LIN {X 0,Y 331.929,Z 1000.191,A -85,B 0,C 180,E1 23009.158,E2 23009.158} C_VEL
LIN {X 0,Y 336.667,Z 1013.449,A -85,B 0,C 180,E1 23012.773,E2 23012.773} C_VEL
LIN {X 0,Y 338.095,Z 1019.979,A -85,B 0,C 180,E1 23013.863,E2 23013.863} C_VEL
LIN {X 0,Y 332.466,Z 1050.059,A -85,B 0,C 180,E1 23015.679,E2 23015.679} C_VEL
LIN {X 0,Y 325.019,Z 1075.85,A -85,B 0,C 180,E1 23018.168,E2 23018.168} C_VEL
LIN {X 0,Y 315.792,Z 1098.668,A -85,B 0,C 180,E1 23021.521,E2 23021.521} C_VEL
LIN {X 0,Y 310.988,Z 1108.297,A -85,B 0,C 180,E1 23023.502,E2 23023.502} C_VEL
LIN {X 0,Y 302.321,Z 1118.917,A -85,B 0,C 180,E1 23025.58,E2 23025.58} C_VEL
LIN {X 0,Y 294.454,Z 1126.629,A -85,B 0,C 180,E1 23027.603,E2 23027.603} C_VEL
LIN {X 0,Y 293.706,Z 1127.508,A -85,B 0,C 180,E1 23027.959,E2 23027.959} C_VEL
LIN {X 0,Y 286.319,Z 1135.333,A -85,B 0,C 180,E1 23032.421,E2 23032.421} C_VEL
LIN {X 0,Y 280.665,Z 1138.98,A -85,B 0,C 180,E1 23036.917,E2 23036.917} C_VEL
LIN {X 0,Y 277.782,Z 1139.343,A -85,B 0,C 180,E1 23040.003,E2 23040.003} C_VEL
LIN {X 0,Y 274.693,Z 1136.847,A -85,B 0,C 180,E1 23044.737,E2 23044.737} C_VEL
LIN {X 0,Y 272.966,Z 1127.598,A -85,B 0,C 180,E1 23051.175,E2 23051.175} C_VEL
LIN {X 0,Y 273.213,Z 1112.925,A -85,B 0,C 180,E1 23056.884,E2 23056.884} C_VEL
LIN {X 0,Y 274.614,Z 1092.685,A -85,B 0,C 180,E1 23061.997,E2 23061.997} C_VEL
LIN {X 0,Y 276.602,Z 1068.704,A -85,B 0,C 180,E1 23066.137,E2 23066.137} C_VEL
LIN {X 0,Y 278.792,Z 1039.52,A -85,B 0,C 180,E1 23069.486,E2 23069.486} C_VEL
LIN {X 0,Y 280.451,Z 1007.858,A -85,B 0,C 180,E1 23071.663,E2 23071.663} C_VEL
LIN {X 0,Y 280.123,Z 983.5,A -85,B 0,C 180,E1 23072.673,E2 23072.673} C_VEL
LIN {X 0,Y 267.448,Z 923.03,A -85,B 0,C 180,E1 23075.683,E2 23075.683} C_VEL
LIN {X 0,Y 266.889,Z 923.03,A -85,B 0,C 180,E1 23082.804,E2 23082.804} C_VEL
LIN {X 0,Y 266.968,Z 923.03,A -85,B 0,C 180,E1 23091.46,E2 23091.46} C_VEL
LIN {X 0,Y 267.275,Z 923.03,A -85,B 0,C 180,E1 23099.384,E2 23099.384} C_VEL
LIN {X 0,Y 267.761,Z 923.03,A -85,B 0,C 180,E1 23106.703,E2 23106.703} C_VEL
LIN {X 0,Y 268.363,Z 923.03,A -85,B 0,C 180,E1 23113.62,E2 23113.62} C_VEL
LIN {X 0,Y 269.003,Z 923.03,A -85,B 0,C 180,E1 23120.27,E2 23120.27} C_VEL
LIN {X 0,Y 269.819,Z 923.03,A -85,B 0,C 180,E1 23126.762,E2 23126.762} C_VEL
LIN {X 0,Y 269.811,Z 923.03,A -85,B 0,C 180,E1 23133.182,E2 23133.182} C_VEL
LIN {X 0,Y 269.095,Z 923.03,A -85,B 0,C 180,E1 23139.669,E2 23139.669} C_VEL
LIN {X 0,Y 268.337,Z 923.03,A -85,B 0,C 180,E1 23146.786,E2 23146.786} C_VEL
LIN {X 0,Y 267.656,Z 923.03,A -85,B 0,C 180,E1 23155.396,E2 23155.396} C_VEL
LIN {X 0,Y 267.187,Z 923.03,A -85,B 0,C 180,E1 23164.403,E2 23164.403} C_VEL
LIN {X 0,Y 267.237,Z 923.488,A -85,B 0,C 180,E1 23165.586,E2 23165.586} C_VEL
LIN {X 0,Y 284.856,Z 968.437,A -85,B 0,C 180,E1 23170.572,E2 23170.572} C_VEL
LIN {X 0,Y 296.502,Z 1005.612,A -85,B 0,C 180,E1 23174.909,E2 23174.909} C_VEL
LIN {X 0,Y 304.304,Z 1038.041,A -85,B 0,C 180,E1 23179.036,E2 23179.036} C_VEL
LIN {X 0,Y 295.095,Z 1075.692,A -85,B 0,C 180,E1 23183.463,E2 23183.463} C_VEL
LIN {X 0,Y 286.275,Z 1109.373,A -85,B 0,C 180,E1 23189.022,E2 23189.022} C_VEL
LIN {X 0,Y 279.131,Z 1136.473,A -85,B 0,C 180,E1 23195.19,E2 23195.19} C_VEL
LIN {X 0,Y 274.28,Z 1158.137,A -85,B 0,C 180,E1 23201.943,E2 23201.943} C_VEL
LIN {X 0,Y 271.653,Z 1173.928,A -85,B 0,C 180,E1 23208.77,E2 23208.77} C_VEL
LIN {X 0,Y 270.65,Z 1184.291,A -85,B 0,C 180,E1 23215.193,E2 23215.193} C_VEL
LIN {X 0,Y 270.557,Z 1190.919,A -85,B 0,C 180,E1 23221.597,E2 23221.597} C_VEL
LIN {X 0,Y 272.362,Z 1194.634,A -85,B 0,C 180,E1 23229.578,E2 23229.578} C_VEL
LIN {X 0,Y 278.537,Z 1193.012,A -85,B 0,C 180,E1 23238.993,E2 23238.993} C_VEL
LIN {X 0,Y 290.948,Z 1185.504,A -85,B 0,C 180,E1 23247.864,E2 23247.864} C_VEL
LIN {X 0,Y 311.71,Z 1171.475,A -85,B 0,C 180,E1 23256.283,E2 23256.283} C_VEL
LIN {X 0,Y 339.898,Z 1151.742,A -85,B 0,C 180,E1 23263.248,E2 23263.248} C_VEL
LIN {X 0,Y 340.347,Z 1151.495,A -85,B 0,C 180,E1 23263.626,E2 23263.626} C_VEL
LIN {X 0,Y 309.964,Z 1177.069,A -85,B 0,C 180,E1 23270.708,E2 23270.708} C_VEL
LIN {X 0,Y 288.327,Z 1196.897,A -85,B 0,C 180,E1 23279.408,E2 23279.408} C_VEL
LIN {X 0,Y 276.425,Z 1209.235,A -85,B 0,C 180,E1 23288.32,E2 23288.32} C_VEL
LIN {X 0,Y 271.361,Z 1215.518,A -85,B 0,C 180,E1 23297.16,E2 23297.16} C_VEL
LIN {X 0,Y 270.484,Z 1216.446,A -85,B 0,C 180,E1 23303.614,E2 23303.614} C_VEL
LIN {X 0,Y 271.033,Z 1214.048,A -85,B 0,C 180,E1 23310.028,E2 23310.028} C_VEL
LIN {X 0,Y 271.147,Z 1206.707,A -85,B 0,C 180,E1 23317.231,E2 23317.231} C_VEL
LIN {X 0,Y 272.139,Z 1193.796,A -85,B 0,C 180,E1 23324.501,E2 23324.501} C_VEL
LIN {X 0,Y 275.469,Z 1175.838,A -85,B 0,C 180,E1 23332.023,E2 23332.023} C_VEL
LIN {X 0,Y 281.759,Z 1158.597,A -85,B 0,C 180,E1 23338.405,E2 23338.405} C_VEL
LIN {X 0,Y 290.902,Z 1135.195,A -85,B 0,C 180,E1 23344.184,E2 23344.184} C_VEL
LIN {X 0,Y 301.149,Z 1107.507,A -85,B 0,C 180,E1 23348.871,E2 23348.871} C_VEL
LIN {X 0,Y 310.736,Z 1076.284,A -85,B 0,C 180,E1 23352.52,E2 23352.52} C_VEL
LIN {X 0,Y 318.06,Z 1045.689,A -85,B 0,C 180,E1 23354.842,E2 23354.842} C_VEL
LIN {X 0,Y 321.177,Z 1017.496,A -85,B 0,C 180,E1 23359.484,E2 23359.484} C_VEL
LIN {X 0,Y 325.671,Z 998.479,A -85,B 0,C 180,E1 23362.748,E2 23362.748} C_VEL
LIN {X 0,Y 326.577,Z 1000.295,A -85,B 0,C 180,E1 23364.99,E2 23364.99} C_VEL
LIN {X 0,Y 329.513,Z 1007.381,A -85,B 0,C 180,E1 23368.754,E2 23368.754} C_VEL
LIN {X 0,Y 333.618,Z 1020.084,A -85,B 0,C 180,E1 23372.232,E2 23372.232} C_VEL
LIN {X 0,Y 334.133,Z 1023.713,A -85,B 0,C 180,E1 23372.802,E2 23372.802} C_VEL
LIN {X 0,Y 327.641,Z 1054.65,A -85,B 0,C 180,E1 23374.772,E2 23374.772} C_VEL
LIN {X 0,Y 319.445,Z 1080.19,A -85,B 0,C 180,E1 23377.386,E2 23377.386} C_VEL
LIN {X 0,Y 309.736,Z 1101.939,A -85,B 0,C 180,E1 23380.776,E2 23380.776} C_VEL
LIN {X 0,Y 299.636,Z 1119.417,A -85,B 0,C 180,E1 23385.025,E2 23385.025} C_VEL
LIN {X 0,Y 293.706,Z 1127.508,A -85,B 0,C 180,E1 23387.959,E2 23387.959} C_VEL
LIN {X 0,Y 285,Z 1134.232,A -85,B 0,C 180,E1 23390.669,E2 23390.669} C_VEL
LIN {X 0,Y 276.923,Z 1138.639,A -85,B 0,C 180,E1 23393.437,E2 23393.437} C_VEL
LIN {X 0,Y 276.615,Z 1138.783,A -85,B 0,C 180,E1 23393.649,E2 23393.649} C_VEL
LIN {X 0,Y 272.435,Z 1140.471,A -85,B 0,C 180,E1 23397.182,E2 23397.182} C_VEL
LIN {X 0,Y 267.601,Z 1138.671,A -85,B 0,C 180,E1 23403.241,E2 23403.241} C_VEL
LIN {X 0,Y 265.203,Z 1130.248,A -85,B 0,C 180,E1 23409.846,E2 23409.846} C_VEL
LIN {X 0,Y 265.193,Z 1116.066,A -85,B 0,C 180,E1 23415.884,E2 23415.884} C_VEL
LIN {X 0,Y 266.366,Z 1096.688,A -85,B 0,C 180,E1 23421.21,E2 23421.21} C_VEL
LIN {X 0,Y 268.449,Z 1072.024,A -85,B 0,C 180,E1 23425.77,E2 23425.77} C_VEL
LIN {X 0,Y 270.68,Z 1043.898,A -85,B 0,C 180,E1 23429.244,E2 23429.244} C_VEL
LIN {X 0,Y 272.452,Z 1012.551,A -85,B 0,C 180,E1 23431.636,E2 23431.636} C_VEL
LIN {X 0,Y 272.442,Z 985.065,A -85,B 0,C 180,E1 23432.86,E2 23432.86} C_VEL
LIN {X 0,Y 259.474,Z 923.03,A -85,B 0,C 180,E1 23436.06,E2 23436.06} C_VEL
LIN {X 0,Y 258.804,Z 923.03,A -85,B 0,C 180,E1 23445.485,E2 23445.485} C_VEL
LIN {X 0,Y 259.146,Z 923.03,A -85,B 0,C 180,E1 23454.727,E2 23454.727} C_VEL
LIN {X 0,Y 259.491,Z 923.03,A -85,B 0,C 180,E1 23462.203,E2 23462.203} C_VEL
LIN {X 0,Y 260.037,Z 923.03,A -85,B 0,C 180,E1 23469.565,E2 23469.565} C_VEL
LIN {X 0,Y 260.736,Z 923.03,A -85,B 0,C 180,E1 23476.567,E2 23476.567} C_VEL
LIN {X 0,Y 261.406,Z 923.03,A -85,B 0,C 180,E1 23483.332,E2 23483.332} C_VEL
LIN {X 0,Y 262.275,Z 923.03,A -85,B 0,C 180,E1 23489.971,E2 23489.971} C_VEL
LIN {X 0,Y 261.431,Z 923.03,A -85,B 0,C 180,E1 23496.608,E2 23496.608} C_VEL
LIN {X 0,Y 260.78,Z 923.03,A -85,B 0,C 180,E1 23503.371,E2 23503.371} C_VEL
LIN {X 0,Y 259.927,Z 923.03,A -85,B 0,C 180,E1 23511.53,E2 23511.53} C_VEL
LIN {X 0,Y 259.397,Z 923.03,A -85,B 0,C 180,E1 23519.088,E2 23519.088} C_VEL
LIN {X 0,Y 259.318,Z 923.086,A -85,B 0,C 180,E1 23524.435,E2 23524.435} C_VEL
LIN {X 0,Y 277.062,Z 968.601,A -85,B 0,C 180,E1 23529.688,E2 23529.688} C_VEL
LIN {X 0,Y 288.779,Z 1006.071,A -85,B 0,C 180,E1 23534.199,E2 23534.199} C_VEL
LIN {X 0,Y 296.79,Z 1039.197,A -85,B 0,C 180,E1 23538.552,E2 23538.552} C_VEL
LIN {X 0,Y 287.203,Z 1077.68,A -85,B 0,C 180,E1 23543.234,E2 23543.234} C_VEL
LIN {X 0,Y 278.191,Z 1110.858,A -85,B 0,C 180,E1 23548.93,E2 23548.93} C_VEL
LIN {X 0,Y 271.018,Z 1137.732,A -85,B 0,C 180,E1 23555.277,E2 23555.277} C_VEL
LIN {X 0,Y 266.161,Z 1159.171,A -85,B 0,C 180,E1 23562.229,E2 23562.229} C_VEL
LIN {X 0,Y 263.646,Z 1174.786,A -85,B 0,C 180,E1 23569.261,E2 23569.261} C_VEL
LIN {X 0,Y 262.693,Z 1186.038,A -85,B 0,C 180,E1 23576.699,E2 23576.699} C_VEL
LIN {X 0,Y 262.872,Z 1192.09,A -85,B 0,C 180,E1 23583.292,E2 23583.292} C_VEL
LIN {X 0,Y 264.546,Z 1195.014,A -85,B 0,C 180,E1 23589.863,E2 23589.863} C_VEL
LIN {X 0,Y 271.109,Z 1194.076,A -85,B 0,C 180,E1 23599.534,E2 23599.534} C_VEL
LIN {X 0,Y 284.144,Z 1187.266,A -85,B 0,C 180,E1 23608.592,E2 23608.592} C_VEL
LIN {X 0,Y 306.084,Z 1173.939,A -85,B 0,C 180,E1 23617.208,E2 23617.208} C_VEL
LIN {X 0,Y 330.733,Z 1158.343,A -85,B 0,C 180,E1 23623.258,E2 23623.258} C_VEL
LIN {X 0,Y 326.707,Z 1161.53,A -85,B 0,C 180,E1 23624.334,E2 23624.334} C_VEL
LIN {X 0,Y 296.273,Z 1185.355,A -85,B 0,C 180,E1 23632.299,E2 23632.299} C_VEL
LIN {X 0,Y 276.511,Z 1202.18,A -85,B 0,C 180,E1 23641.468,E2 23641.468} C_VEL
LIN {X 0,Y 266.872,Z 1211.523,A -85,B 0,C 180,E1 23650.172,E2 23650.172} C_VEL
LIN {X 0,Y 262.83,Z 1215.856,A -85,B 0,C 180,E1 23660.098,E2 23660.098} C_VEL
LIN {X 0,Y 262.819,Z 1214.905,A -85,B 0,C 180,E1 23666.733,E2 23666.733} C_VEL
LIN {X 0,Y 263.238,Z 1210.404,A -85,B 0,C 180,E1 23673.32,E2 23673.32} C_VEL
LIN {X 0,Y 263.658,Z 1200.247,A -85,B 0,C 180,E1 23680.763,E2 23680.763} C_VEL
LIN {X 0,Y 265.615,Z 1184.147,A -85,B 0,C 180,E1 23688.262,E2 23688.262} C_VEL
LIN {X 0,Y 271.611,Z 1167.354,A -85,B 0,C 180,E1 23696.457,E2 23696.457} C_VEL
LIN {X 0,Y 280.273,Z 1147.648,A -85,B 0,C 180,E1 23702.655,E2 23702.655} C_VEL
LIN {X 0,Y 291.384,Z 1122.108,A -85,B 0,C 180,E1 23708.041,E2 23708.041} C_VEL
LIN {X 0,Y 302.826,Z 1092.653,A -85,B 0,C 180,E1 23712.257,E2 23712.257} C_VEL
LIN {X 0,Y 312.499,Z 1061.306,A -85,B 0,C 180,E1 23715.281,E2 23715.281} C_VEL
LIN {X 0,Y 316.077,Z 1046.644,A -85,B 0,C 180,E1 23716.388,E2 23716.388} C_VEL
LIN {X 0,Y 324.081,Z 1006.301,A -85,B 0,C 180,E1 23723.301,E2 23723.301} C_VEL
LIN {X 0,Y 326.301,Z 1012.419,A -85,B 0,C 180,E1 23727.406,E2 23727.406} C_VEL
LIN {X 0,Y 329.781,Z 1023.242,A -85,B 0,C 180,E1 23730.919,E2 23730.919} C_VEL
LIN {X 0,Y 330.363,Z 1027.639,A -85,B 0,C 180,E1 23731.712,E2 23731.712} C_VEL
LIN {X 0,Y 323.081,Z 1058.968,A -85,B 0,C 180,E1 23733.81,E2 23733.81} C_VEL
LIN {X 0,Y 313.469,Z 1085.522,A -85,B 0,C 180,E1 23736.719,E2 23736.719} C_VEL
LIN {X 0,Y 302.864,Z 1106.8,A -85,B 0,C 180,E1 23740.322,E2 23740.322} C_VEL
LIN {X 0,Y 291.574,Z 1124.038,A -85,B 0,C 180,E1 23744.985,E2 23744.985} C_VEL
LIN {X 0,Y 282.075,Z 1134.615,A -85,B 0,C 180,E1 23749.977,E2 23749.977} C_VEL
LIN {X 0,Y 276.615,Z 1138.783,A -85,B 0,C 180,E1 23753.649,E2 23753.649} C_VEL
LIN {X 0,Y 268.765,Z 1141.151,A -85,B 0,C 180,E1 23756.9,E2 23756.9} C_VEL
LIN {X 0,Y 262.115,Z 1141.238,A -85,B 0,C 180,E1 23759.882,E2 23759.882} C_VEL
LIN {X 0,Y 261.65,Z 1141.016,A -85,B 0,C 180,E1 23760.346,E2 23760.346} C_VEL
LIN {X 0,Y 258.057,Z 1135.197,A -85,B 0,C 180,E1 23766.729,E2 23766.729} C_VEL
LIN {X 0,Y 257.099,Z 1124.32,A -85,B 0,C 180,E1 23772.737,E2 23772.737} C_VEL
LIN {X 0,Y 257.676,Z 1108.063,A -85,B 0,C 180,E1 23778.354,E2 23778.354} C_VEL
LIN {X 0,Y 259.344,Z 1086.543,A -85,B 0,C 180,E1 23783.391,E2 23783.391} C_VEL
LIN {X 0,Y 261.603,Z 1060.463,A -85,B 0,C 180,E1 23787.527,E2 23787.527} C_VEL
LIN {X 0,Y 263.853,Z 1028.991,A -85,B 0,C 180,E1 23790.742,E2 23790.742} C_VEL
LIN {X 0,Y 265.235,Z 995.781,A -85,B 0,C 180,E1 23792.621,E2 23792.621} C_VEL
LIN {X 0,Y 263.388,Z 979.844,A -85,B 0,C 180,E1 23793.352,E2 23793.352} C_VEL
LIN {X 0,Y 251.526,Z 923.03,A -85,B 0,C 180,E1 23796.438,E2 23796.438} C_VEL
LIN {X 0,Y 250.817,Z 923.03,A -85,B 0,C 180,E1 23806.305,E2 23806.305} C_VEL
LIN {X 0,Y 250.982,Z 923.03,A -85,B 0,C 180,E1 23812.947,E2 23812.947} C_VEL
LIN {X 0,Y 251.519,Z 923.03,A -85,B 0,C 180,E1 23821.242,E2 23821.242} C_VEL
LIN {X 0,Y 252.045,Z 923.03,A -85,B 0,C 180,E1 23828.887,E2 23828.887} C_VEL
LIN {X 0,Y 252.732,Z 923.03,A -85,B 0,C 180,E1 23836.133,E2 23836.133} C_VEL
LIN {X 0,Y 253.469,Z 923.03,A -85,B 0,C 180,E1 23843.122,E2 23843.122} C_VEL
LIN {X 0,Y 254.382,Z 923.03,A -85,B 0,C 180,E1 23849.97,E2 23849.97} C_VEL
LIN {X 0,Y 253.496,Z 923.03,A -85,B 0,C 180,E1 23856.816,E2 23856.816} C_VEL
LIN {X 0,Y 252.777,Z 923.03,A -85,B 0,C 180,E1 23863.802,E2 23863.802} C_VEL
LIN {X 0,Y 252.079,Z 923.03,A -85,B 0,C 180,E1 23871.046,E2 23871.046} C_VEL
LIN {X 0,Y 251.543,Z 923.03,A -85,B 0,C 180,E1 23878.686,E2 23878.686} C_VEL
LIN {X 0,Y 251.403,Z 923.767,A -85,B 0,C 180,E1 23883.288,E2 23883.288} C_VEL
LIN {X 0,Y 268.93,Z 967.865,A -85,B 0,C 180,E1 23888.649,E2 23888.649} C_VEL
LIN {X 0,Y 280.691,Z 1005.121,A -85,B 0,C 180,E1 23893.292,E2 23893.292} C_VEL
LIN {X 0,Y 289.122,Z 1039.954,A -85,B 0,C 180,E1 23898.001,E2 23898.001} C_VEL
LIN {X 0,Y 279.602,Z 1078.239,A -85,B 0,C 180,E1 23902.794,E2 23902.794} C_VEL
LIN {X 0,Y 270.673,Z 1110.396,A -85,B 0,C 180,E1 23908.437,E2 23908.437} C_VEL
LIN {X 0,Y 263.284,Z 1137.463,A -85,B 0,C 180,E1 23914.954,E2 23914.954} C_VEL
LIN {X 0,Y 258.297,Z 1159.082,A -85,B 0,C 180,E1 23922.109,E2 23922.109} C_VEL
LIN {X 0,Y 255.614,Z 1175.6,A -85,B 0,C 180,E1 23929.781,E2 23929.781} C_VEL
LIN {X 0,Y 254.799,Z 1185.745,A -85,B 0,C 180,E1 23936.596,E2 23936.596} C_VEL
LIN {X 0,Y 254.993,Z 1192.14,A -85,B 0,C 180,E1 23943.394,E2 23943.394} C_VEL
LIN {X 0,Y 256.737,Z 1195.38,A -85,B 0,C 180,E1 23950.167,E2 23950.167} C_VEL
LIN {X 0,Y 263.694,Z 1195.005,A -85,B 0,C 180,E1 23960.107,E2 23960.107} C_VEL
LIN {X 0,Y 277.904,Z 1188.737,A -85,B 0,C 180,E1 23969.607,E2 23969.607} C_VEL
LIN {X 0,Y 300.234,Z 1176.662,A -85,B 0,C 180,E1 23978.061,E2 23978.061} C_VEL
LIN {X 0,Y 320.451,Z 1165.094,A -85,B 0,C 180,E1 23983.072,E2 23983.072} C_VEL
LIN {X 0,Y 321.164,Z 1164.745,A -85,B 0,C 180,E1 23983.479,E2 23983.479} C_VEL
LIN {X 0,Y 290.38,Z 1186.813,A -85,B 0,C 180,E1 23991.308,E2 23991.308} C_VEL
LIN {X 0,Y 269.553,Z 1202.822,A -85,B 0,C 180,E1 24000.661,E2 24000.661} C_VEL
LIN {X 0,Y 259.326,Z 1211.504,A -85,B 0,C 180,E1 24009.569,E2 24009.569} C_VEL
LIN {X 0,Y 254.976,Z 1215.328,A -85,B 0,C 180,E1 24019.79,E2 24019.79} C_VEL
LIN {X 0,Y 254.938,Z 1214.109,A -85,B 0,C 180,E1 24026.632,E2 24026.632} C_VEL
LIN {X 0,Y 255.294,Z 1210.824,A -85,B 0,C 180,E1 24031.726,E2 24031.726} C_VEL
LIN {X 0,Y 255.575,Z 1202.931,A -85,B 0,C 180,E1 24038.53,E2 24038.53} C_VEL
LIN {X 0,Y 256.9,Z 1188.437,A -85,B 0,C 180,E1 24046.254,E2 24046.254} C_VEL
LIN {X 0,Y 257.885,Z 1183.257,A -85,B 0,C 180,E1 24048.83,E2 24048.83} C_VEL
LIN {X 0,Y 262.706,Z 1171.746,A -85,B 0,C 180,E1 24055.586,E2 24055.586} C_VEL
LIN {X 0,Y 271.782,Z 1153.343,A -85,B 0,C 180,E1 24062.384,E2 24062.384} C_VEL
LIN {X 0,Y 283.972,Z 1129.032,A -85,B 0,C 180,E1 24068.244,E2 24068.244} C_VEL
LIN {X 0,Y 297.116,Z 1099.881,A -85,B 0,C 180,E1 24072.892,E2 24072.892} C_VEL
LIN {X 0,Y 308.522,Z 1068.867,A -85,B 0,C 180,E1 24076.171,E2 24076.171} C_VEL
LIN {X 0,Y 313.846,Z 1050.539,A -85,B 0,C 180,E1 24077.622,E2 24077.622} C_VEL
LIN {X 0,Y 322.415,Z 1014.434,A -85,B 0,C 180,E1 24083.78,E2 24083.78} C_VEL
LIN {X 0,Y 324.729,Z 1021.562,A -85,B 0,C 180,E1 24087.84,E2 24087.84} C_VEL
LIN {X 0,Y 326.998,Z 1030.776,A -85,B 0,C 180,E1 24090.551,E2 24090.551} C_VEL
LIN {X 0,Y 319.621,Z 1060.163,A -85,B 0,C 180,E1 24092.554,E2 24092.554} C_VEL
LIN {X 0,Y 309.656,Z 1086.229,A -85,B 0,C 180,E1 24095.394,E2 24095.394} C_VEL
LIN {X 0,Y 298.737,Z 1107.116,A -85,B 0,C 180,E1 24098.878,E2 24098.878} C_VEL
LIN {X 0,Y 286.697,Z 1124.575,A -85,B 0,C 180,E1 24103.546,E2 24103.546} C_VEL
LIN {X 0,Y 275.77,Z 1135.963,A -85,B 0,C 180,E1 24108.947,E2 24108.947} C_VEL
LIN {X 0,Y 268.747,Z 1140.643,A -85,B 0,C 180,E1 24113.547,E2 24113.547} C_VEL
LIN {X 0,Y 264.925,Z 1141.734,A -85,B 0,C 180,E1 24116.734,E2 24116.734} C_VEL
LIN {X 0,Y 261.65,Z 1141.016,A -85,B 0,C 180,E1 24120.346,E2 24120.346} C_VEL
LIN {X 0,Y 255.301,Z 1138.732,A -85,B 0,C 180,E1 24123.927,E2 24123.927} C_VEL
LIN {X 0,Y 249.883,Z 1134.172,A -85,B 0,C 180,E1 24127.583,E2 24127.583} C_VEL
LIN {X 0,Y 249.235,Z 1121.046,A -85,B 0,C 180,E1 24134.039,E2 24134.039} C_VEL
LIN {X 0,Y 250.129,Z 1103.104,A -85,B 0,C 180,E1 24139.705,E2 24139.705} C_VEL
LIN {X 0,Y 252.097,Z 1079.181,A -85,B 0,C 180,E1 24144.813,E2 24144.813} C_VEL
LIN {X 0,Y 254.408,Z 1051.322,A -85,B 0,C 180,E1 24148.794,E2 24148.794} C_VEL
LIN {X 0,Y 256.525,Z 1019.759,A -85,B 0,C 180,E1 24151.604,E2 24151.604} C_VEL
LIN {X 0,Y 256.788,Z 986.82,A -85,B 0,C 180,E1 24153.256,E2 24153.256} C_VEL
LIN {X 0,Y 243.552,Z 923.03,A -85,B 0,C 180,E1 24156.803,E2 24156.803} C_VEL
LIN {X 0,Y 242.925,Z 923.03,A -85,B 0,C 180,E1 24166.786,E2 24166.786} C_VEL
LIN {X 0,Y 243.122,Z 923.03,A -85,B 0,C 180,E1 24175.953,E2 24175.953} C_VEL
LIN {X 0,Y 243.746,Z 923.03,A -85,B 0,C 180,E1 24184.249,E2 24184.249} C_VEL
LIN {X 0,Y 244.348,Z 923.03,A -85,B 0,C 180,E1 24191.957,E2 24191.957} C_VEL
LIN {X 0,Y 245.212,Z 923.03,A -85,B 0,C 180,E1 24200.418,E2 24200.418} C_VEL
LIN {X 0,Y 246.469,Z 923.03,A -85,B 0,C 180,E1 24209.969,E2 24209.969} C_VEL
LIN {X 0,Y 245.278,Z 923.03,A -85,B 0,C 180,E1 24219.672,E2 24219.672} C_VEL
LIN {X 0,Y 244.397,Z 923.03,A -85,B 0,C 180,E1 24227.973,E2 24227.973} C_VEL
LIN {X 0,Y 243.773,Z 923.03,A -85,B 0,C 180,E1 24235.679,E2 24235.679} C_VEL
LIN {X 0,Y 243.406,Z 923.034,A -85,B 0,C 180,E1 24241.998,E2 24241.998} C_VEL
LIN {X 0,Y 261.039,Z 967.845,A -85,B 0,C 180,E1 24247.653,E2 24247.653} C_VEL
LIN {X 0,Y 272.487,Z 1003.964,A -85,B 0,C 180,E1 24252.314,E2 24252.314} C_VEL
LIN {X 0,Y 281.092,Z 1038.968,A -85,B 0,C 180,E1 24257.177,E2 24257.177} C_VEL
LIN {X 0,Y 280.835,Z 1045.041,A -85,B 0,C 180,E1 24257.933,E2 24257.933} C_VEL
LIN {X 0,Y 270.992,Z 1081.931,A -85,B 0,C 180,E1 24262.844,E2 24262.844} C_VEL
LIN {X 0,Y 262.056,Z 1113.66,A -85,B 0,C 180,E1 24268.733,E2 24268.733} C_VEL
LIN {X 0,Y 254.808,Z 1140.051,A -85,B 0,C 180,E1 24275.469,E2 24275.469} C_VEL
LIN {X 0,Y 249.806,Z 1162.19,A -85,B 0,C 180,E1 24283.298,E2 24283.298} C_VEL
LIN {X 0,Y 247.455,Z 1177.878,A -85,B 0,C 180,E1 24291.215,E2 24291.215} C_VEL
LIN {X 0,Y 246.837,Z 1187.353,A -85,B 0,C 180,E1 24298.242,E2 24298.242} C_VEL
LIN {X 0,Y 247.727,Z 1194.32,A -85,B 0,C 180,E1 24307.004,E2 24307.004} C_VEL
LIN {X 0,Y 253.153,Z 1196.514,A -85,B 0,C 180,E1 24317.361,E2 24317.361} C_VEL
LIN {X 0,Y 267.285,Z 1192.106,A -85,B 0,C 180,E1 24328.395,E2 24328.395} C_VEL
LIN {X 0,Y 290.229,Z 1181.399,A -85,B 0,C 180,E1 24337.714,E2 24337.714} C_VEL
LIN {X 0,Y 311.649,Z 1170.506,A -85,B 0,C 180,E1 24343.38,E2 24343.38} C_VEL
LIN {X 0,Y 281.092,Z 1190.602,A -85,B 0,C 180,E1 24351.448,E2 24351.448} C_VEL
LIN {X 0,Y 261.093,Z 1204.525,A -85,B 0,C 180,E1 24360.793,E2 24360.793} C_VEL
LIN {X 0,Y 251.84,Z 1211.5,A -85,B 0,C 180,E1 24368.933,E2 24368.933} C_VEL
LIN {X 0,Y 247.126,Z 1214.801,A -85,B 0,C 180,E1 24379.462,E2 24379.462} C_VEL
LIN {X 0,Y 247.19,Z 1212.291,A -85,B 0,C 180,E1 24388.279,E2 24388.279} C_VEL
LIN {X 0,Y 247.579,Z 1206.19,A -85,B 0,C 180,E1 24395.283,E2 24395.283} C_VEL
LIN {X 0,Y 248.322,Z 1193.974,A -85,B 0,C 180,E1 24403.201,E2 24403.201} C_VEL
LIN {X 0,Y 249.583,Z 1184.808,A -85,B 0,C 180,E1 24407.652,E2 24407.652} C_VEL
LIN {X 0,Y 254.63,Z 1173.769,A -85,B 0,C 180,E1 24415.514,E2 24415.514} C_VEL
LIN {X 0,Y 263.909,Z 1157.191,A -85,B 0,C 180,E1 24422.497,E2 24422.497} C_VEL
LIN {X 0,Y 276.411,Z 1135.154,A -85,B 0,C 180,E1 24428.483,E2 24428.483} C_VEL
LIN {X 0,Y 290.608,Z 1107.784,A -85,B 0,C 180,E1 24433.385,E2 24433.385} C_VEL
LIN {X 0,Y 303.831,Z 1077.572,A -85,B 0,C 180,E1 24436.934,E2 24436.934} C_VEL
LIN {X 0,Y 311.796,Z 1054.113,A -85,B 0,C 180,E1 24438.905,E2 24438.905} C_VEL
LIN {X 0,Y 320.468,Z 1023.636,A -85,B 0,C 180,E1 24444.172,E2 24444.172} C_VEL
LIN {X 0,Y 322.016,Z 1027.434,A -85,B 0,C 180,E1 24446.85,E2 24446.85} C_VEL
LIN {X 0,Y 323.62,Z 1035.205,A -85,B 0,C 180,E1 24449.442,E2 24449.442} C_VEL
LIN {X 0,Y 315.849,Z 1063.274,A -85,B 0,C 180,E1 24451.421,E2 24451.421} C_VEL
LIN {X 0,Y 305.095,Z 1089.192,A -85,B 0,C 180,E1 24454.321,E2 24454.321} C_VEL
LIN {X 0,Y 292.874,Z 1110.614,A -85,B 0,C 180,E1 24458.059,E2 24458.059} C_VEL
LIN {X 0,Y 280.341,Z 1127.128,A -85,B 0,C 180,E1 24462.758,E2 24462.758} C_VEL
LIN {X 0,Y 269.58,Z 1137.364,A -85,B 0,C 180,E1 24467.869,E2 24467.869} C_VEL
LIN {X 0,Y 260.958,Z 1142.294,A -85,B 0,C 180,E1 24473.353,E2 24473.353} C_VEL
LIN {X 0,Y 253.969,Z 1141.972,A -85,B 0,C 180,E1 24480.004,E2 24480.004} C_VEL
LIN {X 0,Y 250.49,Z 1136.678,A -85,B 0,C 180,E1 24485.751,E2 24485.751} C_VEL
LIN {X 0,Y 249.883,Z 1134.172,A -85,B 0,C 180,E1 24487.583,E2 24487.583} C_VEL
LIN {X 0,Y 246.856,Z 1129.438,A -85,B 0,C 180,E1 24490.324,E2 24490.324} C_VEL
LIN {X 0,Y 241.449,Z 1120.296,A -85,B 0,C 180,E1 24494.267,E2 24494.267} C_VEL
LIN {X 0,Y 241.382,Z 1119.09,A -85,B 0,C 180,E1 24494.708,E2 24494.708} C_VEL
LIN {X 0,Y 242.467,Z 1099.82,A -85,B 0,C 180,E1 24500.537,E2 24500.537} C_VEL
LIN {X 0,Y 244.602,Z 1074.815,A -85,B 0,C 180,E1 24505.627,E2 24505.627} C_VEL
LIN {X 0,Y 246.948,Z 1046.516,A -85,B 0,C 180,E1 24509.47,E2 24509.47} C_VEL
LIN {X 0,Y 248.9,Z 1014.919,A -85,B 0,C 180,E1 24512.121,E2 24512.121} C_VEL
LIN {X 0,Y 249.083,Z 988.336,A -85,B 0,C 180,E1 24513.434,E2 24513.434} C_VEL
LIN {X 0,Y 235.594,Z 923.03,A -85,B 0,C 180,E1 24517.186,E2 24517.186} C_VEL
LIN {X 0,Y 234.913,Z 923.03,A -85,B 0,C 180,E1 24525.044,E2 24525.044} C_VEL
LIN {X 0,Y 235.051,Z 923.03,A -85,B 0,C 180,E1 24530.491,E2 24530.491} C_VEL
LIN {X 0,Y 235.33,Z 923.03,A -85,B 0,C 180,E1 24539.055,E2 24539.055} C_VEL
LIN {X 0,Y 235.967,Z 923.03,A -85,B 0,C 180,E1 24547.371,E2 24547.371} C_VEL
LIN {X 0,Y 236.734,Z 923.03,A -85,B 0,C 180,E1 24555.175,E2 24555.175} C_VEL
LIN {X 0,Y 237.56,Z 923.03,A -85,B 0,C 180,E1 24562.659,E2 24562.659} C_VEL
LIN {X 0,Y 238.564,Z 923.03,A -85,B 0,C 180,E1 24569.968,E2 24569.968} C_VEL
LIN {X 0,Y 237.594,Z 923.03,A -85,B 0,C 180,E1 24577.275,E2 24577.275} C_VEL
LIN {X 0,Y 236.53,Z 923.03,A -85,B 0,C 180,E1 24586.593,E2 24586.593} C_VEL
LIN {X 0,Y 235.769,Z 923.03,A -85,B 0,C 180,E1 24596.187,E2 24596.187} C_VEL
LIN {X 0,Y 235.551,Z 923.629,A -85,B 0,C 180,E1 24600.735,E2 24600.735} C_VEL
LIN {X 0,Y 253.155,Z 967.719,A -85,B 0,C 180,E1 24606.607,E2 24606.607} C_VEL
LIN {X 0,Y 264.663,Z 1003.667,A -85,B 0,C 180,E1 24611.421,E2 24611.421} C_VEL
LIN {X 0,Y 273.29,Z 1039.083,A -85,B 0,C 180,E1 24616.482,E2 24616.482} C_VEL
LIN {X 0,Y 273.36,Z 1045.938,A -85,B 0,C 180,E1 24617.395,E2 24617.395} C_VEL
LIN {X 0,Y 263.107,Z 1083.357,A -85,B 0,C 180,E1 24622.546,E2 24622.546} C_VEL
LIN {X 0,Y 253.718,Z 1115.794,A -85,B 0,C 180,E1 24628.819,E2 24628.819} C_VEL
LIN {X 0,Y 246.086,Z 1143.503,A -85,B 0,C 180,E1 24636.32,E2 24636.32} C_VEL
LIN {X 0,Y 241.305,Z 1165.035,A -85,B 0,C 180,E1 24644.561,E2 24644.561} C_VEL
LIN {X 0,Y 239.296,Z 1179.973,A -85,B 0,C 180,E1 24652.741,E2 24652.741} C_VEL
LIN {X 0,Y 239.023,Z 1188.877,A -85,B 0,C 180,E1 24659.996,E2 24659.996} C_VEL
LIN {X 0,Y 239.868,Z 1194.417,A -85,B 0,C 180,E1 24667.234,E2 24667.234} C_VEL
LIN {X 0,Y 245.619,Z 1197.243,A -85,B 0,C 180,E1 24677.911,E2 24677.911} C_VEL
LIN {X 0,Y 258.178,Z 1194.355,A -85,B 0,C 180,E1 24687.916,E2 24687.916} C_VEL
LIN {X 0,Y 278.237,Z 1186.524,A -85,B 0,C 180,E1 24696.68,E2 24696.68} C_VEL
LIN {X 0,Y 300.731,Z 1176.399,A -85,B 0,C 180,E1 24702.896,E2 24702.896} C_VEL
LIN {X 0,Y 301.355,Z 1176.22,A -85,B 0,C 180,E1 24703.431,E2 24703.431} C_VEL
LIN {X 0,Y 273.591,Z 1192.964,A -85,B 0,C 180,E1 24710.951,E2 24710.951} C_VEL
LIN {X 0,Y 252.011,Z 1206.435,A -85,B 0,C 180,E1 24721.372,E2 24721.372} C_VEL
LIN {X 0,Y 241.862,Z 1213.032,A -85,B 0,C 180,E1 24731.832,E2 24731.832} C_VEL
LIN {X 0,Y 239.304,Z 1214.176,A -85,B 0,C 180,E1 24739.114,E2 24739.114} C_VEL
LIN {X 0,Y 239.362,Z 1211.331,A -85,B 0,C 180,E1 24748.223,E2 24748.223} C_VEL
LIN {X 0,Y 239.76,Z 1204.833,A -85,B 0,C 180,E1 24755.456,E2 24755.456} C_VEL
LIN {X 0,Y 240.471,Z 1193.088,A -85,B 0,C 180,E1 24763.185,E2 24763.185} C_VEL
LIN {X 0,Y 241.604,Z 1185.012,A -85,B 0,C 180,E1 24767.314,E2 24767.314} C_VEL
LIN {X 0,Y 246.487,Z 1175.445,A -85,B 0,C 180,E1 24775.444,E2 24775.444} C_VEL
LIN {X 0,Y 256.627,Z 1159.505,A -85,B 0,C 180,E1 24783.034,E2 24783.034} C_VEL
LIN {X 0,Y 270.595,Z 1137.747,A -85,B 0,C 180,E1 24789.468,E2 24789.468} C_VEL
LIN {X 0,Y 285.961,Z 1111.423,A -85,B 0,C 180,E1 24794.472,E2 24794.472} C_VEL
LIN {X 0,Y 300.724,Z 1081.573,A -85,B 0,C 180,E1 24798.132,E2 24798.132} C_VEL
LIN {X 0,Y 309.949,Z 1057.762,A -85,B 0,C 180,E1 24800.195,E2 24800.195} C_VEL
LIN {X 0,Y 318.932,Z 1031.737,A -85,B 0,C 180,E1 24804.719,E2 24804.719} C_VEL
LIN {X 0,Y 320.347,Z 1038.77,A -85,B 0,C 180,E1 24808.007,E2 24808.007} C_VEL
LIN {X 0,Y 320.031,Z 1041.425,A -85,B 0,C 180,E1 24808.405,E2 24808.405} C_VEL
LIN {X 0,Y 310.565,Z 1070.832,A -85,B 0,C 180,E1 24810.669,E2 24810.669} C_VEL
LIN {X 0,Y 298.727,Z 1095.823,A -85,B 0,C 180,E1 24813.733,E2 24813.733} C_VEL
LIN {X 0,Y 285.992,Z 1115.604,A -85,B 0,C 180,E1 24817.572,E2 24817.572} C_VEL
LIN {X 0,Y 273.155,Z 1130.621,A -85,B 0,C 180,E1 24822.29,E2 24822.29} C_VEL
LIN {X 0,Y 263.472,Z 1138.82,A -85,B 0,C 180,E1 24826.741,E2 24826.741} C_VEL
LIN {X 0,Y 253.142,Z 1143.869,A -85,B 0,C 180,E1 24833.147,E2 24833.147} C_VEL
LIN {X 0,Y 245.992,Z 1142.556,A -85,B 0,C 180,E1 24840.004,E2 24840.004} C_VEL
LIN {X 0,Y 242.491,Z 1136.49,A -85,B 0,C 180,E1 24845.976,E2 24845.976} C_VEL
LIN {X 0,Y 241.335,Z 1124.666,A -85,B 0,C 180,E1 24852.485,E2 24852.485} C_VEL
LIN {X 0,Y 241.382,Z 1119.09,A -85,B 0,C 180,E1 24854.708,E2 24854.708} C_VEL
LIN {X 0,Y 239.2,Z 1111.674,A -85,B 0,C 180,E1 24857.218,E2 24857.218} C_VEL
LIN {X 0,Y 234.733,Z 1098.871,A -85,B 0,C 180,E1 24860.75,E2 24860.75} C_VEL
LIN {X 0,Y 234.739,Z 1097.288,A -85,B 0,C 180,E1 24861.137,E2 24861.137} C_VEL
LIN {X 0,Y 236.856,Z 1072.914,A -85,B 0,C 180,E1 24866.02,E2 24866.02} C_VEL
LIN {X 0,Y 239.23,Z 1044.328,A -85,B 0,C 180,E1 24869.856,E2 24869.856} C_VEL
LIN {X 0,Y 241.134,Z 1012.092,A -85,B 0,C 180,E1 24872.48,E2 24872.48} C_VEL
LIN {X 0,Y 241.082,Z 988.367,A -85,B 0,C 180,E1 24873.664,E2 24873.664} C_VEL
LIN {X 0,Y 227.666,Z 923.03,A -85,B 0,C 180,E1 24877.432,E2 24877.432} C_VEL
LIN {X 0,Y 226.88,Z 923.03,A -85,B 0,C 180,E1 24888.198,E2 24888.198} C_VEL
LIN {X 0,Y 227.327,Z 923.03,A -85,B 0,C 180,E1 24897.838,E2 24897.838} C_VEL
LIN {X 0,Y 227.957,Z 923.03,A -85,B 0,C 180,E1 24906.529,E2 24906.529} C_VEL
LIN {X 0,Y 228.737,Z 923.03,A -85,B 0,C 180,E1 24914.645,E2 24914.645} C_VEL
LIN {X 0,Y 229.588,Z 923.03,A -85,B 0,C 180,E1 24922.403,E2 24922.403} C_VEL
LIN {X 0,Y 230.648,Z 923.03,A -85,B 0,C 180,E1 24929.967,E2 24929.967} C_VEL
LIN {X 0,Y 229.406,Z 923.03,A -85,B 0,C 180,E1 24938.841,E2 24938.841} C_VEL
LIN {X 0,Y 228.777,Z 923.03,A -85,B 0,C 180,E1 24945.284,E2 24945.284} C_VEL
LIN {X 0,Y 227.966,Z 923.03,A -85,B 0,C 180,E1 24953.397,E2 24953.397} C_VEL
LIN {X 0,Y 227.703,Z 923.082,A -85,B 0,C 180,E1 24959.314,E2 24959.314} C_VEL
LIN {X 0,Y 245.294,Z 967.572,A -85,B 0,C 180,E1 24965.506,E2 24965.506} C_VEL
LIN {X 0,Y 257.053,Z 1004.47,A -85,B 0,C 180,E1 24970.639,E2 24970.639} C_VEL
LIN {X 0,Y 265.669,Z 1040.187,A -85,B 0,C 180,E1 24975.925,E2 24975.925} C_VEL
LIN {X 0,Y 265.628,Z 1047.608,A -85,B 0,C 180,E1 24976.944,E2 24976.944} C_VEL
LIN {X 0,Y 255.4,Z 1084.097,A -85,B 0,C 180,E1 24982.127,E2 24982.127} C_VEL
LIN {X 0,Y 246.056,Z 1115.638,A -85,B 0,C 180,E1 24988.399,E2 24988.399} C_VEL
LIN {X 0,Y 238.194,Z 1143.617,A -85,B 0,C 180,E1 24996.166,E2 24996.166} C_VEL
LIN {X 0,Y 233.603,Z 1163.877,A -85,B 0,C 180,E1 25004.039,E2 25004.039} C_VEL
LIN {X 0,Y 231.442,Z 1179.289,A -85,B 0,C 180,E1 25012.493,E2 25012.493} C_VEL
LIN {X 0,Y 231.127,Z 1188.554,A -85,B 0,C 180,E1 25019.996,E2 25019.996} C_VEL
LIN {X 0,Y 232.014,Z 1194.415,A -85,B 0,C 180,E1 25027.481,E2 25027.481} C_VEL
LIN {X 0,Y 238.112,Z 1197.844,A -85,B 0,C 180,E1 25038.496,E2 25038.496} C_VEL
LIN {X 0,Y 251.289,Z 1195.675,A -85,B 0,C 180,E1 25048.751,E2 25048.751} C_VEL
LIN {X 0,Y 276.305,Z 1187.097,A -85,B 0,C 180,E1 25058.967,E2 25058.967} C_VEL
LIN {X 0,Y 291.239,Z 1181.137,A -85,B 0,C 180,E1 25062.911,E2 25062.911} C_VEL
LIN {X 0,Y 291.129,Z 1181.336,A -85,B 0,C 180,E1 25063.436,E2 25063.436} C_VEL
LIN {X 0,Y 262.362,Z 1197.12,A -85,B 0,C 180,E1 25071.787,E2 25071.787} C_VEL
LIN {X 0,Y 242.684,Z 1208.151,A -85,B 0,C 180,E1 25082.199,E2 25082.199} C_VEL
LIN {X 0,Y 234.27,Z 1212.677,A -85,B 0,C 180,E1 25091.221,E2 25091.221} C_VEL
LIN {X 0,Y 231.504,Z 1213.474,A -85,B 0,C 180,E1 25098.742,E2 25098.742} C_VEL
LIN {X 0,Y 231.528,Z 1210.285,A -85,B 0,C 180,E1 25108.163,E2 25108.163} C_VEL
LIN {X 0,Y 231.952,Z 1203.41,A -85,B 0,C 180,E1 25115.64,E2 25115.64} C_VEL
LIN {X 0,Y 232.614,Z 1192.424,A -85,B 0,C 180,E1 25123.004,E2 25123.004} C_VEL
LIN {X 0,Y 233.587,Z 1184.93,A -85,B 0,C 180,E1 25126.957,E2 25126.957} C_VEL
LIN {X 0,Y 238.341,Z 1176.803,A -85,B 0,C 180,E1 25135.371,E2 25135.371} C_VEL
LIN {X 0,Y 248.608,Z 1162.622,A -85,B 0,C 180,E1 25143.197,E2 25143.197} C_VEL
LIN {X 0,Y 262.872,Z 1142.943,A -85,B 0,C 180,E1 25149.789,E2 25149.789} C_VEL
LIN {X 0,Y 279.8,Z 1117.523,A -85,B 0,C 180,E1 25155.173,E2 25155.173} C_VEL
LIN {X 0,Y 296.349,Z 1088.246,A -85,B 0,C 180,E1 25159.084,E2 25159.084} C_VEL
LIN {X 0,Y 308.205,Z 1061.827,A -85,B 0,C 180,E1 25161.422,E2 25161.422} C_VEL
LIN {X 0,Y 317.04,Z 1040.405,A -85,B 0,C 180,E1 25165.389,E2 25165.389} C_VEL
LIN {X 0,Y 317.356,Z 1044.423,A -85,B 0,C 180,E1 25167.113,E2 25167.113} C_VEL
LIN {X 0,Y 307.014,Z 1074.244,A -85,B 0,C 180,E1 25169.501,E2 25169.501} C_VEL
LIN {X 0,Y 294.682,Z 1098.328,A -85,B 0,C 180,E1 25172.519,E2 25172.519} C_VEL
LIN {X 0,Y 280.809,Z 1118.297,A -85,B 0,C 180,E1 25176.498,E2 25176.498} C_VEL
LIN {X 0,Y 267.778,Z 1132.315,A -85,B 0,C 180,E1 25181.07,E2 25181.07} C_VEL
LIN {X 0,Y 255.963,Z 1141.26,A -85,B 0,C 180,E1 25186.345,E2 25186.345} C_VEL
LIN {X 0,Y 245.325,Z 1145.281,A -85,B 0,C 180,E1 25192.927,E2 25192.927} C_VEL
LIN {X 0,Y 241.222,Z 1144.966,A -85,B 0,C 180,E1 25196.412,E2 25196.412} C_VEL
LIN {X 0,Y 236.133,Z 1140.583,A -85,B 0,C 180,E1 25202.755,E2 25202.755} C_VEL
LIN {X 0,Y 233.729,Z 1131.066,A -85,B 0,C 180,E1 25209.305,E2 25209.305} C_VEL
LIN {X 0,Y 233.674,Z 1115.313,A -85,B 0,C 180,E1 25215.956,E2 25215.956} C_VEL
LIN {X 0,Y 234.739,Z 1097.288,A -85,B 0,C 180,E1 25221.137,E2 25221.137} C_VEL
LIN {X 0,Y 231.852,Z 1084.392,A -85,B 0,C 180,E1 25223.971,E2 25223.971} C_VEL
LIN {X 0,Y 229.17,Z 1070.324,A -85,B 0,C 180,E1 25226.521,E2 25226.521} C_VEL
LIN {X 0,Y 231.582,Z 1040.793,A -85,B 0,C 180,E1 25230.382,E2 25230.382} C_VEL
LIN {X 0,Y 233.453,Z 1008.923,A -85,B 0,C 180,E1 25232.852,E2 25232.852} C_VEL
LIN {X 0,Y 233.139,Z 988.951,A -85,B 0,C 180,E1 25233.867,E2 25233.867} C_VEL
LIN {X 0,Y 219.659,Z 923.03,A -85,B 0,C 180,E1 25237.95,E2 25237.95} C_VEL
LIN {X 0,Y 218.875,Z 923.03,A -85,B 0,C 180,E1 25249.421,E2 25249.421} C_VEL
LIN {X 0,Y 219.195,Z 923.03,A -85,B 0,C 180,E1 25256.491,E2 25256.491} C_VEL
LIN {X 0,Y 219.86,Z 923.03,A -85,B 0,C 180,E1 25265.61,E2 25265.61} C_VEL
LIN {X 0,Y 220.694,Z 923.03,A -85,B 0,C 180,E1 25274.07,E2 25274.07} C_VEL
LIN {X 0,Y 221.626,Z 923.03,A -85,B 0,C 180,E1 25282.128,E2 25282.128} C_VEL
LIN {X 0,Y 222.73,Z 923.03,A -85,B 0,C 180,E1 25289.966,E2 25289.966} C_VEL
LIN {X 0,Y 221.679,Z 923.03,A -85,B 0,C 180,E1 25297.8,E2 25297.8} C_VEL
LIN {X 0,Y 220.619,Z 923.03,A -85,B 0,C 180,E1 25306.467,E2 25306.467} C_VEL
LIN {X 0,Y 219.76,Z 923.03,A -85,B 0,C 180,E1 25316.623,E2 25316.623} C_VEL
LIN {X 0,Y 219.818,Z 923.339,A -85,B 0,C 180,E1 25317.857,E2 25317.857} C_VEL
LIN {X 0,Y 237.722,Z 967.986,A -85,B 0,C 180,E1 25324.438,E2 25324.438} C_VEL
LIN {X 0,Y 249.601,Z 1005.613,A -85,B 0,C 180,E1 25329.888,E2 25329.888} C_VEL
LIN {X 0,Y 257.812,Z 1040.093,A -85,B 0,C 180,E1 25335.155,E2 25335.155} C_VEL
LIN {X 0,Y 258.283,Z 1047.95,A -85,B 0,C 180,E1 25336.314,E2 25336.314} C_VEL
LIN {X 0,Y 247.845,Z 1084.212,A -85,B 0,C 180,E1 25341.597,E2 25341.597} C_VEL
LIN {X 0,Y 238.41,Z 1115.345,A -85,B 0,C 180,E1 25347.934,E2 25347.934} C_VEL
LIN {X 0,Y 230.453,Z 1143.044,A -85,B 0,C 180,E1 25355.802,E2 25355.802} C_VEL
LIN {X 0,Y 225.513,Z 1164.614,A -85,B 0,C 180,E1 25364.449,E2 25364.449} C_VEL
LIN {X 0,Y 223.457,Z 1179.923,A -85,B 0,C 180,E1 25373.199,E2 25373.199} C_VEL
LIN {X 0,Y 223.268,Z 1190.006,A -85,B 0,C 180,E1 25381.935,E2 25381.935} C_VEL
LIN {X 0,Y 225.607,Z 1196.39,A -85,B 0,C 180,E1 25391.588,E2 25391.588} C_VEL
LIN {X 0,Y 234.317,Z 1198.464,A -85,B 0,C 180,E1 25402.76,E2 25402.76} C_VEL
LIN {X 0,Y 254.361,Z 1194.429,A -85,B 0,C 180,E1 25414.354,E2 25414.354} C_VEL
LIN {X 0,Y 282.023,Z 1185.399,A -85,B 0,C 180,E1 25423.211,E2 25423.211} C_VEL
LIN {X 0,Y 254.315,Z 1199.045,A -85,B 0,C 180,E1 25431.442,E2 25431.442} C_VEL
LIN {X 0,Y 235.615,Z 1208.251,A -85,B 0,C 180,E1 25441.289,E2 25441.289} C_VEL
LIN {X 0,Y 226.678,Z 1212.327,A -85,B 0,C 180,E1 25450.568,E2 25450.568} C_VEL
LIN {X 0,Y 223.322,Z 1211.923,A -85,B 0,C 180,E1 25462.258,E2 25462.258} C_VEL
LIN {X 0,Y 224.079,Z 1207.819,A -85,B 0,C 180,E1 25470.034,E2 25470.034} C_VEL
LIN {X 0,Y 224.277,Z 1199.476,A -85,B 0,C 180,E1 25477.778,E2 25477.778} C_VEL
LIN {X 0,Y 225.611,Z 1184.564,A -85,B 0,C 180,E1 25486.572,E2 25486.572} C_VEL
LIN {X 0,Y 230.203,Z 1177.826,A -85,B 0,C 180,E1 25495.291,E2 25495.291} C_VEL
LIN {X 0,Y 240.544,Z 1165.291,A -85,B 0,C 180,E1 25503.379,E2 25503.379} C_VEL
LIN {X 0,Y 256.084,Z 1146.374,A -85,B 0,C 180,E1 25510.507,E2 25510.507} C_VEL
LIN {X 0,Y 273.656,Z 1123.046,A -85,B 0,C 180,E1 25515.911,E2 25515.911} C_VEL
LIN {X 0,Y 291.357,Z 1095.434,A -85,B 0,C 180,E1 25519.941,E2 25519.941} C_VEL
LIN {X 0,Y 307.001,Z 1064.587,A -85,B 0,C 180,E1 25522.869,E2 25522.869} C_VEL
LIN {X 0,Y 313.933,Z 1049.974,A -85,B 0,C 180,E1 25525.552,E2 25525.552} C_VEL
LIN {X 0,Y 314.324,Z 1049.994,A -85,B 0,C 180,E1 25526.058,E2 25526.058} C_VEL
LIN {X 0,Y 303.527,Z 1078.105,A -85,B 0,C 180,E1 25528.339,E2 25528.339} C_VEL
LIN {X 0,Y 289.627,Z 1102.795,A -85,B 0,C 180,E1 25531.573,E2 25531.573} C_VEL
LIN {X 0,Y 275.828,Z 1120.936,A -85,B 0,C 180,E1 25535.363,E2 25535.363} C_VEL
LIN {X 0,Y 260.635,Z 1135.647,A -85,B 0,C 180,E1 25540.53,E2 25540.53} C_VEL
LIN {X 0,Y 248.456,Z 1143.592,A -85,B 0,C 180,E1 25545.924,E2 25545.924} C_VEL
LIN {X 0,Y 237.486,Z 1146.554,A -85,B 0,C 180,E1 25552.693,E2 25552.693} C_VEL
LIN {X 0,Y 230.002,Z 1143.374,A -85,B 0,C 180,E1 25560.004,E2 25560.004} C_VEL
LIN {X 0,Y 226.15,Z 1133.646,A -85,B 0,C 180,E1 25567.684,E2 25567.684} C_VEL
LIN {X 0,Y 225.582,Z 1119.729,A -85,B 0,C 180,E1 25574.218,E2 25574.218} C_VEL
LIN {X 0,Y 226.63,Z 1100.52,A -85,B 0,C 180,E1 25580.277,E2 25580.277} C_VEL
LIN {X 0,Y 228.78,Z 1075.251,A -85,B 0,C 180,E1 25585.691,E2 25585.691} C_VEL
LIN {X 0,Y 229.17,Z 1070.324,A -85,B 0,C 180,E1 25586.521,E2 25586.521} C_VEL
LIN {X 0,Y 226.496,Z 1055.418,A -85,B 0,C 180,E1 25588.754,E2 25588.754} C_VEL
LIN {X 0,Y 223.778,Z 1039.687,A -85,B 0,C 180,E1 25590.643,E2 25590.643} C_VEL
LIN {X 0,Y 225.665,Z 1007.105,A -85,B 0,C 180,E1 25593.165,E2 25593.165} C_VEL
LIN {X 0,Y 225.146,Z 988.955,A -85,B 0,C 180,E1 25594.115,E2 25594.115} C_VEL
LIN {X 0,Y 211.686,Z 923.03,A -85,B 0,C 180,E1 25598.207,E2 25598.207} C_VEL
LIN {X 0,Y 210.968,Z 923.03,A -85,B 0,C 180,E1 25609.818,E2 25609.818} C_VEL
LIN {X 0,Y 211.407,Z 923.03,A -85,B 0,C 180,E1 25619.938,E2 25619.938} C_VEL
LIN {X 0,Y 212.203,Z 923.03,A -85,B 0,C 180,E1 25629.106,E2 25629.106} C_VEL
LIN {X 0,Y 213.129,Z 923.03,A -85,B 0,C 180,E1 25637.684,E2 25637.684} C_VEL
LIN {X 0,Y 214.207,Z 923.03,A -85,B 0,C 180,E1 25645.919,E2 25645.919} C_VEL
LIN {X 0,Y 214.81,Z 923.03,A -85,B 0,C 180,E1 25649.965,E2 25649.965} C_VEL
LIN {X 0,Y 213.698,Z 923.03,A -85,B 0,C 180,E1 25658.093,E2 25658.093} C_VEL
LIN {X 0,Y 212.712,Z 923.03,A -85,B 0,C 180,E1 25666.47,E2 25666.47} C_VEL
LIN {X 0,Y 211.905,Z 923.796,A -85,B 0,C 180,E1 25676.335,E2 25676.335} C_VEL
LIN {X 0,Y 229.134,Z 965.818,A -85,B 0,C 180,E1 25682.918,E2 25682.918} C_VEL
LIN {X 0,Y 241.004,Z 1002.893,A -85,B 0,C 180,E1 25688.497,E2 25688.497} C_VEL
LIN {X 0,Y 249.924,Z 1039.254,A -85,B 0,C 180,E1 25694.238,E2 25694.238} C_VEL
LIN {X 0,Y 250.8,Z 1048.651,A -85,B 0,C 180,E1 25695.709,E2 25695.709} C_VEL
LIN {X 0,Y 239.87,Z 1085.602,A -85,B 0,C 180,E1 25701.272,E2 25701.272} C_VEL
LIN {X 0,Y 229.781,Z 1118.252,A -85,B 0,C 180,E1 25708.253,E2 25708.253} C_VEL
LIN {X 0,Y 221.988,Z 1145.449,A -85,B 0,C 180,E1 25716.499,E2 25716.499} C_VEL
LIN {X 0,Y 217.464,Z 1165.193,A -85,B 0,C 180,E1 25724.831,E2 25724.831} C_VEL
LIN {X 0,Y 215.533,Z 1180.512,A -85,B 0,C 180,E1 25733.959,E2 25733.959} C_VEL
LIN {X 0,Y 215.406,Z 1189.623,A -85,B 0,C 180,E1 25742.006,E2 25742.006} C_VEL
LIN {X 0,Y 217.837,Z 1196.532,A -85,B 0,C 180,E1 25752.007,E2 25752.007} C_VEL
LIN {X 0,Y 227.041,Z 1199.232,A -85,B 0,C 180,E1 25763.532,E2 25763.532} C_VEL
LIN {X 0,Y 244.353,Z 1196.872,A -85,B 0,C 180,E1 25773.814,E2 25773.814} C_VEL
LIN {X 0,Y 270.985,Z 1189.681,A -85,B 0,C 180,E1 25782.701,E2 25782.701} C_VEL
LIN {X 0,Y 271.531,Z 1189.627,A -85,B 0,C 180,E1 25783.267,E2 25783.267} C_VEL
LIN {X 0,Y 240.698,Z 1203.251,A -85,B 0,C 180,E1 25793.43,E2 25793.43} C_VEL
LIN {X 0,Y 222.17,Z 1210.935,A -85,B 0,C 180,E1 25805.955,E2 25805.955} C_VEL
LIN {X 0,Y 215.922,Z 1212.025,A -85,B 0,C 180,E1 25817.918,E2 25817.918} C_VEL
LIN {X 0,Y 215.923,Z 1207.943,A -85,B 0,C 180,E1 25828.03,E2 25828.03} C_VEL
LIN {X 0,Y 216.365,Z 1200.484,A -85,B 0,C 180,E1 25836.048,E2 25836.048} C_VEL
LIN {X 0,Y 217.237,Z 1188.036,A -85,B 0,C 180,E1 25844.221,E2 25844.221} C_VEL
LIN {X 0,Y 217.762,Z 1183.76,A -85,B 0,C 180,E1 25846.668,E2 25846.668} C_VEL
LIN {X 0,Y 222.948,Z 1177.613,A -85,B 0,C 180,E1 25856.175,E2 25856.175} C_VEL
LIN {X 0,Y 233.951,Z 1165.985,A -85,B 0,C 180,E1 25864.45,E2 25864.45} C_VEL
LIN {X 0,Y 250.318,Z 1148.331,A -85,B 0,C 180,E1 25871.644,E2 25871.644} C_VEL
LIN {X 0,Y 268.679,Z 1126.561,A -85,B 0,C 180,E1 25877.018,E2 25877.018} C_VEL
LIN {X 0,Y 288.294,Z 1099.088,A -85,B 0,C 180,E1 25881.206,E2 25881.206} C_VEL
LIN {X 0,Y 304.947,Z 1069.871,A -85,B 0,C 180,E1 25883.905,E2 25883.905} C_VEL
LIN {X 0,Y 309.007,Z 1062.175,A -85,B 0,C 180,E1 25885.392,E2 25885.392} C_VEL
LIN {X 0,Y 296.416,Z 1088.938,A -85,B 0,C 180,E1 25887.937,E2 25887.937} C_VEL
LIN {X 0,Y 280.959,Z 1112.063,A -85,B 0,C 180,E1 25891.493,E2 25891.493} C_VEL
LIN {X 0,Y 265.518,Z 1129.017,A -85,B 0,C 180,E1 25895.807,E2 25895.807} C_VEL
LIN {X 0,Y 249.678,Z 1141.321,A -85,B 0,C 180,E1 25901.478,E2 25901.478} C_VEL
LIN {X 0,Y 240.936,Z 1145.726,A -85,B 0,C 180,E1 25905.475,E2 25905.475} C_VEL
LIN {X 0,Y 229.642,Z 1147.718,A -85,B 0,C 180,E1 25912.442,E2 25912.442} C_VEL
LIN {X 0,Y 221.991,Z 1143.508,A -85,B 0,C 180,E1 25920.004,E2 25920.004} C_VEL
LIN {X 0,Y 218.448,Z 1134.526,A -85,B 0,C 180,E1 25926.957,E2 25926.957} C_VEL
LIN {X 0,Y 217.706,Z 1120.185,A -85,B 0,C 180,E1 25933.859,E2 25933.859} C_VEL
LIN {X 0,Y 218.718,Z 1100.397,A -85,B 0,C 180,E1 25940.213,E2 25940.213} C_VEL
LIN {X 0,Y 220.831,Z 1076.053,A -85,B 0,C 180,E1 25945.581,E2 25945.581} C_VEL
LIN {X 0,Y 223.328,Z 1046.144,A -85,B 0,C 180,E1 25949.939,E2 25949.939} C_VEL
LIN {X 0,Y 223.778,Z 1039.687,A -85,B 0,C 180,E1 25950.643,E2 25950.643} C_VEL
LIN {X 0,Y 222.217,Z 1027.453,A -85,B 0,C 180,E1 25951.831,E2 25951.831} C_VEL
LIN {X 0,Y 217.872,Z 1008.857,A -85,B 0,C 180,E1 25953.248,E2 25953.248} C_VEL
LIN {X 0,Y 217.82,Z 1006.706,A -85,B 0,C 180,E1 25953.368,E2 25953.368} C_VEL
LIN {X 0,Y 217.253,Z 989.442,A -85,B 0,C 180,E1 25954.315,E2 25954.315} C_VEL
LIN {X 0,Y 203.653,Z 923.03,A -85,B 0,C 180,E1 25958.731,E2 25958.731} C_VEL
LIN {X 0,Y 202.953,Z 923.03,A -85,B 0,C 180,E1 25968.128,E2 25968.128} C_VEL
LIN {X 0,Y 203.235,Z 923.03,A -85,B 0,C 180,E1 25974.881,E2 25974.881} C_VEL
LIN {X 0,Y 203.706,Z 923.03,A -85,B 0,C 180,E1 25983.532,E2 25983.532} C_VEL
LIN {X 0,Y 204.775,Z 923.03,A -85,B 0,C 180,E1 25993.615,E2 25993.615} C_VEL
LIN {X 0,Y 205.653,Z 923.03,A -85,B 0,C 180,E1 26001.513,E2 26001.513} C_VEL
LIN {X 0,Y 206.914,Z 923.03,A -85,B 0,C 180,E1 26009.963,E2 26009.963} C_VEL
LIN {X 0,Y 205.707,Z 923.03,A -85,B 0,C 180,E1 26018.41,E2 26018.41} C_VEL
LIN {X 0,Y 204.67,Z 923.03,A -85,B 0,C 180,E1 26027.136,E2 26027.136} C_VEL
LIN {X 0,Y 204.004,Z 923.03,A -85,B 0,C 180,E1 26034.575,E2 26034.575} C_VEL
LIN {X 0,Y 221.293,Z 965.65,A -85,B 0,C 180,E1 26041.62,E2 26041.62} C_VEL
LIN {X 0,Y 233.273,Z 1002.95,A -85,B 0,C 180,E1 26047.482,E2 26047.482} C_VEL
LIN {X 0,Y 241.963,Z 1038.811,A -85,B 0,C 180,E1 26053.342,E2 26053.342} C_VEL
LIN {X 0,Y 243.27,Z 1049.571,A -85,B 0,C 180,E1 26055.118,E2 26055.118} C_VEL
LIN {X 0,Y 232.331,Z 1085.622,A -85,B 0,C 180,E1 26060.694,E2 26060.694} C_VEL
LIN {X 0,Y 222.239,Z 1117.482,A -85,B 0,C 180,E1 26067.676,E2 26067.676} C_VEL
LIN {X 0,Y 214.345,Z 1144.382,A -85,B 0,C 180,E1 26075.956,E2 26075.956} C_VEL
LIN {X 0,Y 209.396,Z 1165.948,A -85,B 0,C 180,E1 26085.365,E2 26085.365} C_VEL
LIN {X 0,Y 207.605,Z 1181.052,A -85,B 0,C 180,E1 26094.775,E2 26094.775} C_VEL
LIN {X 0,Y 207.682,Z 1191,A -85,B 0,C 180,E1 26104.168,E2 26104.168} C_VEL
LIN {X 0,Y 210.092,Z 1196.518,A -85,B 0,C 180,E1 26112.457,E2 26112.457} C_VEL
LIN {X 0,Y 219.799,Z 1199.871,A -85,B 0,C 180,E1 26124.357,E2 26124.357} C_VEL
LIN {X 0,Y 237.926,Z 1198.205,A -85,B 0,C 180,E1 26134.857,E2 26134.857} C_VEL
LIN {X 0,Y 260.751,Z 1193.206,A -85,B 0,C 180,E1 26142.599,E2 26142.599} C_VEL
LIN {X 0,Y 261.319,Z 1193.181,A -85,B 0,C 180,E1 26143.25,E2 26143.25} C_VEL
LIN {X 0,Y 230.781,Z 1205.093,A -85,B 0,C 180,E1 26153.938,E2 26153.938} C_VEL
LIN {X 0,Y 212.957,Z 1211.17,A -85,B 0,C 180,E1 26167.276,E2 26167.276} C_VEL
LIN {X 0,Y 208.168,Z 1211.112,A -85,B 0,C 180,E1 26177.461,E2 26177.461} C_VEL
LIN {X 0,Y 208.108,Z 1206.743,A -85,B 0,C 180,E1 26187.956,E2 26187.956} C_VEL
LIN {X 0,Y 208.555,Z 1200.097,A -85,B 0,C 180,E1 26195.233,E2 26195.233} C_VEL
LIN {X 0,Y 209.367,Z 1187.332,A -85,B 0,C 180,E1 26203.982,E2 26203.982} C_VEL
LIN {X 0,Y 209.95,Z 1182.795,A -85,B 0,C 180,E1 26206.768,E2 26206.768} C_VEL
LIN {X 0,Y 213.897,Z 1178.896,A -85,B 0,C 180,E1 26215.116,E2 26215.116} C_VEL
LIN {X 0,Y 224.361,Z 1169.436,A -85,B 0,C 180,E1 26223.793,E2 26223.793} C_VEL
LIN {X 0,Y 241.13,Z 1153.683,A -85,B 0,C 180,E1 26231.604,E2 26231.604} C_VEL
LIN {X 0,Y 261.188,Z 1132.727,A -85,B 0,C 180,E1 26237.569,E2 26237.569} C_VEL
LIN {X 0,Y 281.34,Z 1108.113,A -85,B 0,C 180,E1 26241.806,E2 26241.806} C_VEL
LIN {X 0,Y 299.518,Z 1080.814,A -85,B 0,C 180,E1 26244.667,E2 26244.667} C_VEL
LIN {X 0,Y 301.401,Z 1077.709,A -85,B 0,C 180,E1 26245.125,E2 26245.125} C_VEL
LIN {X 0,Y 287.644,Z 1101.055,A -85,B 0,C 180,E1 26247.87,E2 26247.87} C_VEL
LIN {X 0,Y 272.203,Z 1120.284,A -85,B 0,C 180,E1 26251.396,E2 26251.396} C_VEL
LIN {X 0,Y 256.955,Z 1134.474,A -85,B 0,C 180,E1 26255.695,E2 26255.695} C_VEL
LIN {X 0,Y 244.344,Z 1143.01,A -85,B 0,C 180,E1 26260.119,E2 26260.119} C_VEL
LIN {X 0,Y 233.386,Z 1147.739,A -85,B 0,C 180,E1 26264.994,E2 26264.994} C_VEL
LIN {X 0,Y 221.771,Z 1148.688,A -85,B 0,C 180,E1 26272.172,E2 26272.172} C_VEL
LIN {X 0,Y 213.957,Z 1143.5,A -85,B 0,C 180,E1 26280.004,E2 26280.004} C_VEL
LIN {X 0,Y 210.476,Z 1133.602,A -85,B 0,C 180,E1 26287.222,E2 26287.222} C_VEL
LIN {X 0,Y 209.858,Z 1117.378,A -85,B 0,C 180,E1 26294.696,E2 26294.696} C_VEL
LIN {X 0,Y 211.072,Z 1097.077,A -85,B 0,C 180,E1 26300.98,E2 26300.98} C_VEL
LIN {X 0,Y 213.3,Z 1071.323,A -85,B 0,C 180,E1 26306.433,E2 26306.433} C_VEL
LIN {X 0,Y 215.845,Z 1040.889,A -85,B 0,C 180,E1 26310.652,E2 26310.652} C_VEL
LIN {X 0,Y 217.778,Z 1008.082,A -85,B 0,C 180,E1 26313.293,E2 26313.293} C_VEL
LIN {X 0,Y 217.82,Z 1006.706,A -85,B 0,C 180,E1 26313.368,E2 26313.368} C_VEL
LIN {X 0,Y 214.829,Z 994.28,A -85,B 0,C 180,E1 26314.124,E2 26314.124} C_VEL
LIN {X 0,Y 206.055,Z 974.272,A -85,B 0,C 180,E1 26315.501,E2 26315.501} C_VEL
LIN {X 0,Y 195.7,Z 923.03,A -85,B 0,C 180,E1 26319.091,E2 26319.091} C_VEL
LIN {X 0,Y 194.966,Z 923.03,A -85,B 0,C 180,E1 26331.635,E2 26331.635} C_VEL
LIN {X 0,Y 195.434,Z 923.03,A -85,B 0,C 180,E1 26338.277,E2 26338.277} C_VEL
LIN {X 0,Y 196.141,Z 923.03,A -85,B 0,C 180,E1 26347.605,E2 26347.605} C_VEL
LIN {X 0,Y 197.113,Z 923.03,A -85,B 0,C 180,E1 26356.665,E2 26356.665} C_VEL
LIN {X 0,Y 198.283,Z 923.03,A -85,B 0,C 180,E1 26365.591,E2 26365.591} C_VEL
LIN {X 0,Y 198.989,Z 923.03,A -85,B 0,C 180,E1 26369.962,E2 26369.962} C_VEL
LIN {X 0,Y 197.72,Z 923.03,A -85,B 0,C 180,E1 26378.752,E2 26378.752} C_VEL
LIN {X 0,Y 196.599,Z 923.03,A -85,B 0,C 180,E1 26387.863,E2 26387.863} C_VEL
LIN {X 0,Y 196.203,Z 923.846,A -85,B 0,C 180,E1 26392.874,E2 26392.874} C_VEL
LIN {X 0,Y 212.747,Z 963.507,A -85,B 0,C 180,E1 26399.917,E2 26399.917} C_VEL
LIN {X 0,Y 225.093,Z 1001.397,A -85,B 0,C 180,E1 26406.153,E2 26406.153} C_VEL
LIN {X 0,Y 233.911,Z 1037.421,A -85,B 0,C 180,E1 26412.242,E2 26412.242} C_VEL
LIN {X 0,Y 235.759,Z 1050.398,A -85,B 0,C 180,E1 26414.487,E2 26414.487} C_VEL
LIN {X 0,Y 224.524,Z 1086.399,A -85,B 0,C 180,E1 26420.244,E2 26420.244} C_VEL
LIN {X 0,Y 214.324,Z 1118.007,A -85,B 0,C 180,E1 26427.418,E2 26427.418} C_VEL
LIN {X 0,Y 205.976,Z 1146.265,A -85,B 0,C 180,E1 26436.575,E2 26436.575} C_VEL
LIN {X 0,Y 201.359,Z 1166.523,A -85,B 0,C 180,E1 26445.879,E2 26445.879} C_VEL
LIN {X 0,Y 199.652,Z 1181.54,A -85,B 0,C 180,E1 26455.655,E2 26455.655} C_VEL
LIN {X 0,Y 199.813,Z 1190.55,A -85,B 0,C 180,E1 26464.333,E2 26464.333} C_VEL
LIN {X 0,Y 203.796,Z 1197.769,A -85,B 0,C 180,E1 26475.597,E2 26475.597} C_VEL
LIN {X 0,Y 218.011,Z 1200.616,A -85,B 0,C 180,E1 26489.02,E2 26489.02} C_VEL
LIN {X 0,Y 239.703,Z 1198.292,A -85,B 0,C 180,E1 26499.075,E2 26499.075} C_VEL
LIN {X 0,Y 250.554,Z 1196.218,A -85,B 0,C 180,E1 26502.483,E2 26502.483} C_VEL
LIN {X 0,Y 251.152,Z 1196.241,A -85,B 0,C 180,E1 26503.234,E2 26503.234} C_VEL
LIN {X 0,Y 220.911,Z 1206.496,A -85,B 0,C 180,E1 26514.495,E2 26514.495} C_VEL
LIN {X 0,Y 207.613,Z 1210.277,A -85,B 0,C 180,E1 26524.149,E2 26524.149} C_VEL
LIN {X 0,Y 200.422,Z 1210.188,A -85,B 0,C 180,E1 26536.968,E2 26536.968} C_VEL
LIN {X 0,Y 200.322,Z 1205.367,A -85,B 0,C 180,E1 26547.877,E2 26547.877} C_VEL
LIN {X 0,Y 200.783,Z 1198.385,A -85,B 0,C 180,E1 26555.436,E2 26555.436} C_VEL
LIN {X 0,Y 201.589,Z 1185.894,A -85,B 0,C 180,E1 26564.138,E2 26564.138} C_VEL
LIN {X 0,Y 202.167,Z 1181.603,A -85,B 0,C 180,E1 26566.874,E2 26566.874} C_VEL
LIN {X 0,Y 206.601,Z 1178.336,A -85,B 0,C 180,E1 26576.069,E2 26576.069} C_VEL
LIN {X 0,Y 219.348,Z 1168.45,A -85,B 0,C 180,E1 26585.882,E2 26585.882} C_VEL
LIN {X 0,Y 236.815,Z 1153.864,A -85,B 0,C 180,E1 26593.349,E2 26593.349} C_VEL
LIN {X 0,Y 257.578,Z 1134.336,A -85,B 0,C 180,E1 26599.092,E2 26599.092} C_VEL
LIN {X 0,Y 279.029,Z 1110.444,A -85,B 0,C 180,E1 26603.273,E2 26603.273} C_VEL
LIN {X 0,Y 291.335,Z 1094.297,A -85,B 0,C 180,E1 26605.215,E2 26605.215} C_VEL
LIN {X 0,Y 274.316,Z 1116.607,A -85,B 0,C 180,E1 26608.668,E2 26608.668} C_VEL
LIN {X 0,Y 256.259,Z 1133.637,A -85,B 0,C 180,E1 26613.182,E2 26613.182} C_VEL
LIN {X 0,Y 239.171,Z 1144.716,A -85,B 0,C 180,E1 26618.702,E2 26618.702} C_VEL
LIN {X 0,Y 225.825,Z 1149.619,A -85,B 0,C 180,E1 26624.479,E2 26624.479} C_VEL
LIN {X 0,Y 213.763,Z 1149.455,A -85,B 0,C 180,E1 26631.97,E2 26631.97} C_VEL
LIN {X 0,Y 205.921,Z 1143.199,A -85,B 0,C 180,E1 26640.005,E2 26640.005} C_VEL
LIN {X 0,Y 202.374,Z 1131.467,A -85,B 0,C 180,E1 26648.053,E2 26648.053} C_VEL
LIN {X 0,Y 202.099,Z 1114.279,A -85,B 0,C 180,E1 26655.564,E2 26655.564} C_VEL
LIN {X 0,Y 203.407,Z 1093.271,A -85,B 0,C 180,E1 26661.81,E2 26661.81} C_VEL
LIN {X 0,Y 205.71,Z 1067.469,A -85,B 0,C 180,E1 26667.108,E2 26667.108} C_VEL
LIN {X 0,Y 208.214,Z 1036.781,A -85,B 0,C 180,E1 26671.203,E2 26671.203} C_VEL
LIN {X 0,Y 210.103,Z 1003.191,A -85,B 0,C 180,E1 26673.75,E2 26673.75} C_VEL
LIN {X 0,Y 209.153,Z 989.13,A -85,B 0,C 180,E1 26674.565,E2 26674.565} C_VEL
LIN {X 0,Y 206.055,Z 974.272,A -85,B 0,C 180,E1 26675.501,E2 26675.501} C_VEL
LIN {X 0,Y 198.838,Z 958.803,A -85,B 0,C 180,E1 26676.663,E2 26676.663} C_VEL
LIN {X 0,Y 191.666,Z 943.342,A -85,B 0,C 180,E1 26677.908,E2 26677.908} C_VEL
LIN {X 0,Y 187.716,Z 923.03,A -85,B 0,C 180,E1 26679.415,E2 26679.415} C_VEL
LIN {X 0,Y 186.89,Z 923.03,A -85,B 0,C 180,E1 26689.647,E2 26689.647} C_VEL
LIN {X 0,Y 187.574,Z 923.03,A -85,B 0,C 180,E1 26701.051,E2 26701.051} C_VEL
LIN {X 0,Y 188.519,Z 923.03,A -85,B 0,C 180,E1 26711.258,E2 26711.258} C_VEL
LIN {X 0,Y 189.64,Z 923.03,A -85,B 0,C 180,E1 26720.79,E2 26720.79} C_VEL
LIN {X 0,Y 191.09,Z 923.03,A -85,B 0,C 180,E1 26729.96,E2 26729.96} C_VEL
LIN {X 0,Y 189.712,Z 923.03,A -85,B 0,C 180,E1 26739.125,E2 26739.125} C_VEL
LIN {X 0,Y 188.549,Z 923.03,A -85,B 0,C 180,E1 26748.653,E2 26748.653} C_VEL
LIN {X 0,Y 188.356,Z 923.884,A -85,B 0,C 180,E1 26750.932,E2 26750.932} C_VEL
LIN {X 0,Y 204.745,Z 962.567,A -85,B 0,C 180,E1 26758.321,E2 26758.321} C_VEL
LIN {X 0,Y 217.01,Z 1000.069,A -85,B 0,C 180,E1 26764.803,E2 26764.803} C_VEL
LIN {X 0,Y 226.036,Z 1037.024,A -85,B 0,C 180,E1 26771.263,E2 26771.263} C_VEL
LIN {X 0,Y 228.164,Z 1051.371,A -85,B 0,C 180,E1 26773.859,E2 26773.859} C_VEL
LIN {X 0,Y 216.52,Z 1087.914,A -85,B 0,C 180,E1 26779.928,E2 26779.928} C_VEL
LIN {X 0,Y 205.859,Z 1120.321,A -85,B 0,C 180,E1 26787.667,E2 26787.667} C_VEL
LIN {X 0,Y 197.847,Z 1146.849,A -85,B 0,C 180,E1 26796.735,E2 26796.735} C_VEL
LIN {X 0,Y 193.32,Z 1167.042,A -85,B 0,C 180,E1 26806.433,E2 26806.433} C_VEL
LIN {X 0,Y 191.762,Z 1181.983,A -85,B 0,C 180,E1 26816.607,E2 26816.607} C_VEL
LIN {X 0,Y 192.332,Z 1191.842,A -85,B 0,C 180,E1 26826.763,E2 26826.763} C_VEL
LIN {X 0,Y 197.253,Z 1198.46,A -85,B 0,C 180,E1 26837.839,E2 26837.839} C_VEL
LIN {X 0,Y 211.143,Z 1201.4,A -85,B 0,C 180,E1 26850.059,E2 26850.059} C_VEL
LIN {X 0,Y 238.3,Z 1199.116,A -85,B 0,C 180,E1 26861.74,E2 26861.74} C_VEL
LIN {X 0,Y 240.327,Z 1198.774,A -85,B 0,C 180,E1 26862.363,E2 26862.363} C_VEL
LIN {X 0,Y 240.952,Z 1198.847,A -85,B 0,C 180,E1 26863.216,E2 26863.216} C_VEL
LIN {X 0,Y 211.079,Z 1207.475,A -85,B 0,C 180,E1 26875.108,E2 26875.108} C_VEL
LIN {X 0,Y 196.716,Z 1210.214,A -85,B 0,C 180,E1 26887.457,E2 26887.457} C_VEL
LIN {X 0,Y 192.081,Z 1207.736,A -85,B 0,C 180,E1 26900.989,E2 26900.989} C_VEL
LIN {X 0,Y 192.944,Z 1202.301,A -85,B 0,C 180,E1 26910.04,E2 26910.04} C_VEL
LIN {X 0,Y 193.227,Z 1192.374,A -85,B 0,C 180,E1 26919.037,E2 26919.037} C_VEL
LIN {X 0,Y 194.422,Z 1180.229,A -85,B 0,C 180,E1 26926.985,E2 26926.985} C_VEL
LIN {X 0,Y 199.376,Z 1177.615,A -85,B 0,C 180,E1 26937.089,E2 26937.089} C_VEL
LIN {X 0,Y 212.92,Z 1168.755,A -85,B 0,C 180,E1 26947.144,E2 26947.144} C_VEL
LIN {X 0,Y 231.242,Z 1155.297,A -85,B 0,C 180,E1 26954.667,E2 26954.667} C_VEL
LIN {X 0,Y 254.145,Z 1135.909,A -85,B 0,C 180,E1 26960.661,E2 26960.661} C_VEL
LIN {X 0,Y 277.37,Z 1112.211,A -85,B 0,C 180,E1 26964.845,E2 26964.845} C_VEL
LIN {X 0,Y 279.971,Z 1109.307,A -85,B 0,C 180,E1 26965.506,E2 26965.506} C_VEL
LIN {X 0,Y 262.128,Z 1127.772,A -85,B 0,C 180,E1 26969.232,E2 26969.232} C_VEL
LIN {X 0,Y 243.296,Z 1141.678,A -85,B 0,C 180,E1 26974.234,E2 26974.234} C_VEL
LIN {X 0,Y 225.778,Z 1149.646,A -85,B 0,C 180,E1 26980.454,E2 26980.454} C_VEL
LIN {X 0,Y 211.64,Z 1151.48,A -85,B 0,C 180,E1 26987.636,E2 26987.636} C_VEL
LIN {X 0,Y 201.388,Z 1147.298,A -85,B 0,C 180,E1 26995.701,E2 26995.701} C_VEL
LIN {X 0,Y 195.537,Z 1136.88,A -85,B 0,C 180,E1 27004.437,E2 27004.437} C_VEL
LIN {X 0,Y 194.113,Z 1121.605,A -85,B 0,C 180,E1 27012.352,E2 27012.352} C_VEL
LIN {X 0,Y 194.931,Z 1101.129,A -85,B 0,C 180,E1 27019.531,E2 27019.531} C_VEL
LIN {X 0,Y 197.087,Z 1075.854,A -85,B 0,C 180,E1 27025.554,E2 27025.554} C_VEL
LIN {X 0,Y 199.621,Z 1046.706,A -85,B 0,C 180,E1 27030.17,E2 27030.17} C_VEL
LIN {X 0,Y 201.788,Z 1014.822,A -85,B 0,C 180,E1 27033.214,E2 27033.214} C_VEL
LIN {X 0,Y 201.914,Z 993.056,A -85,B 0,C 180,E1 27034.532,E2 27034.532} C_VEL
LIN {X 0,Y 191.666,Z 943.342,A -85,B 0,C 180,E1 27037.908,E2 27037.908} C_VEL
LIN {X 0,Y 185.57,Z 933.536,A -85,B 0,C 180,E1 27038.816,E2 27038.816} C_VEL
LIN {X 0,Y 179.876,Z 924.467,A -85,B 0,C 180,E1 27039.718,E2 27039.718} C_VEL
LIN {X 0,Y 179.76,Z 923.775,A -85,B 0,C 180,E1 27039.785,E2 27039.785} C_VEL
LIN {X 0,Y 178.996,Z 923.03,A -85,B 0,C 180,E1 27049.453,E2 27049.453} C_VEL
LIN {X 0,Y 179.375,Z 923.03,A -85,B 0,C 180,E1 27059.592,E2 27059.592} C_VEL
LIN {X 0,Y 180.081,Z 923.03,A -85,B 0,C 180,E1 27067.387,E2 27067.387} C_VEL
LIN {X 0,Y 181.031,Z 923.03,A -85,B 0,C 180,E1 27075.456,E2 27075.456} C_VEL
LIN {X 0,Y 182.367,Z 923.03,A -85,B 0,C 180,E1 27085.206,E2 27085.206} C_VEL
LIN {X 0,Y 183.16,Z 923.03,A -85,B 0,C 180,E1 27089.958,E2 27089.958} C_VEL
LIN {X 0,Y 181.697,Z 923.03,A -85,B 0,C 180,E1 27099.531,E2 27099.531} C_VEL
LIN {X 0,Y 180.653,Z 923.552,A -85,B 0,C 180,E1 27108.838,E2 27108.838} C_VEL
LIN {X 0,Y 197.228,Z 962.92,A -85,B 0,C 180,E1 27116.859,E2 27116.859} C_VEL
LIN {X 0,Y 209.389,Z 1000.386,A -85,B 0,C 180,E1 27123.648,E2 27123.648} C_VEL
LIN {X 0,Y 218.225,Z 1036.752,A -85,B 0,C 180,E1 27130.276,E2 27130.276} C_VEL
LIN {X 0,Y 220.629,Z 1052.146,A -85,B 0,C 180,E1 27133.176,E2 27133.176} C_VEL
LIN {X 0,Y 208.871,Z 1088.242,A -85,B 0,C 180,E1 27139.369,E2 27139.369} C_VEL
LIN {X 0,Y 197.982,Z 1120.441,A -85,B 0,C 180,E1 27147.326,E2 27147.326} C_VEL
LIN {X 0,Y 189.605,Z 1147.884,A -85,B 0,C 180,E1 27157.132,E2 27157.132} C_VEL
LIN {X 0,Y 185.165,Z 1168.491,A -85,B 0,C 180,E1 27167.642,E2 27167.642} C_VEL
LIN {X 0,Y 183.923,Z 1182.369,A -85,B 0,C 180,E1 27177.641,E2 27177.641} C_VEL
LIN {X 0,Y 184.497,Z 1191.325,A -85,B 0,C 180,E1 27187.052,E2 27187.052} C_VEL
LIN {X 0,Y 189.719,Z 1198.4,A -85,B 0,C 180,E1 27198.573,E2 27198.573} C_VEL
LIN {X 0,Y 204.321,Z 1201.964,A -85,B 0,C 180,E1 27211.173,E2 27211.173} C_VEL
LIN {X 0,Y 231.125,Z 1200.763,A -85,B 0,C 180,E1 27222.573,E2 27222.573} C_VEL
LIN {X 0,Y 229.427,Z 1201.361,A -85,B 0,C 180,E1 27223.626,E2 27223.626} C_VEL
LIN {X 0,Y 202.058,Z 1207.912,A -85,B 0,C 180,E1 27235.341,E2 27235.341} C_VEL
LIN {X 0,Y 189.377,Z 1209.448,A -85,B 0,C 180,E1 27246.533,E2 27246.533} C_VEL
LIN {X 0,Y 184.329,Z 1206.424,A -85,B 0,C 180,E1 27260.606,E2 27260.606} C_VEL
LIN {X 0,Y 185.219,Z 1200.677,A -85,B 0,C 180,E1 27270.041,E2 27270.041} C_VEL
LIN {X 0,Y 185.486,Z 1190.394,A -85,B 0,C 180,E1 27279.418,E2 27279.418} C_VEL
LIN {X 0,Y 186.7,Z 1178.662,A -85,B 0,C 180,E1 27287.103,E2 27287.103} C_VEL
LIN {X 0,Y 192.23,Z 1176.819,A -85,B 0,C 180,E1 27298.184,E2 27298.184} C_VEL
LIN {X 0,Y 206.613,Z 1168.954,A -85,B 0,C 180,E1 27308.48,E2 27308.48} C_VEL
LIN {X 0,Y 225.781,Z 1156.612,A -85,B 0,C 180,E1 27316.054,E2 27316.054} C_VEL
LIN {X 0,Y 249.457,Z 1138.62,A -85,B 0,C 180,E1 27321.993,E2 27321.993} C_VEL
LIN {X 0,Y 267.23,Z 1122.746,A -85,B 0,C 180,E1 27325.153,E2 27325.153} C_VEL
LIN {X 0,Y 268.423,Z 1121.573,A -85,B 0,C 180,E1 27325.744,E2 27325.744} C_VEL
LIN {X 0,Y 249.164,Z 1137.414,A -85,B 0,C 180,E1 27329.982,E2 27329.982} C_VEL
LIN {X 0,Y 231.672,Z 1147.266,A -85,B 0,C 180,E1 27334.919,E2 27334.919} C_VEL
LIN {X 0,Y 218.405,Z 1151.717,A -85,B 0,C 180,E1 27339.765,E2 27339.765} C_VEL
LIN {X 0,Y 203.861,Z 1152.444,A -85,B 0,C 180,E1 27347.156,E2 27347.156} C_VEL
LIN {X 0,Y 193.384,Z 1147.252,A -85,B 0,C 180,E1 27355.523,E2 27355.523} C_VEL
LIN {X 0,Y 187.531,Z 1135.697,A -85,B 0,C 180,E1 27364.627,E2 27364.627} C_VEL
LIN {X 0,Y 186.274,Z 1118.849,A -85,B 0,C 180,E1 27373.071,E2 27373.071} C_VEL
LIN {X 0,Y 187.267,Z 1097.806,A -85,B 0,C 180,E1 27380.232,E2 27380.232} C_VEL
LIN {X 0,Y 189.553,Z 1071.516,A -85,B 0,C 180,E1 27386.329,E2 27386.329} C_VEL
LIN {X 0,Y 192.102,Z 1042.142,A -85,B 0,C 180,E1 27390.796,E2 27390.796} C_VEL
LIN {X 0,Y 194.096,Z 1009.971,A -85,B 0,C 180,E1 27393.688,E2 27393.688} C_VEL
LIN {X 0,Y 193.779,Z 992.606,A -85,B 0,C 180,E1 27394.772,E2 27394.772} C_VEL
LIN {X 0,Y 179.76,Z 923.775,A -85,B 0,C 180,E1 27399.785,E2 27399.785} C_VEL
LIN {X 0,Y 178.16,Z 919.964,A -85,B 0,C 180,E1 27401.017,E2 27401.017} C_VEL
LIN {X 0,Y 174.427,Z 919.253,A -85,B 0,C 180,E1 27404.206,E2 27404.206} C_VEL
LIN {X 0,Y 170.907,Z 923.03,A -85,B 0,C 180,E1 27410.887,E2 27410.887} C_VEL
LIN {X 0,Y 171.488,Z 923.03,A -85,B 0,C 180,E1 27421.795,E2 27421.795} C_VEL
LIN {X 0,Y 172.354,Z 923.03,A -85,B 0,C 180,E1 27429.425,E2 27429.425} C_VEL
LIN {X 0,Y 173.606,Z 923.03,A -85,B 0,C 180,E1 27439.931,E2 27439.931} C_VEL
LIN {X 0,Y 175.233,Z 923.03,A -85,B 0,C 180,E1 27449.956,E2 27449.956} C_VEL
LIN {X 0,Y 173.665,Z 923.03,A -85,B 0,C 180,E1 27459.976,E2 27459.976} C_VEL
LIN {X 0,Y 172.934,Z 923.656,A -85,B 0,C 180,E1 27466.593,E2 27466.593} C_VEL
LIN {X 0,Y 189.222,Z 962.161,A -85,B 0,C 180,E1 27475.056,E2 27475.056} C_VEL
LIN {X 0,Y 200.708,Z 997.123,A -85,B 0,C 180,E1 27481.756,E2 27481.756} C_VEL
LIN {X 0,Y 209.481,Z 1032.246,A -85,B 0,C 180,E1 27488.422,E2 27488.422} C_VEL
LIN {X 0,Y 213.102,Z 1053.044,A -85,B 0,C 180,E1 27492.482,E2 27492.482} C_VEL
LIN {X 0,Y 200.828,Z 1089.606,A -85,B 0,C 180,E1 27499.01,E2 27499.01} C_VEL
LIN {X 0,Y 189.59,Z 1122.042,A -85,B 0,C 180,E1 27507.447,E2 27507.447} C_VEL
LIN {X 0,Y 181.445,Z 1148.355,A -85,B 0,C 180,E1 27517.34,E2 27517.34} C_VEL
LIN {X 0,Y 177.271,Z 1168.05,A -85,B 0,C 180,E1 27527.778,E2 27527.778} C_VEL
LIN {X 0,Y 176.084,Z 1182.692,A -85,B 0,C 180,E1 27538.765,E2 27538.765} C_VEL
LIN {X 0,Y 177.287,Z 1192.52,A -85,B 0,C 180,E1 27549.81,E2 27549.81} C_VEL
LIN {X 0,Y 186.244,Z 1200.2,A -85,B 0,C 180,E1 27563.928,E2 27563.928} C_VEL
LIN {X 0,Y 204.817,Z 1202.942,A -85,B 0,C 180,E1 27576.167,E2 27576.167} C_VEL
LIN {X 0,Y 220.896,Z 1202.482,A -85,B 0,C 180,E1 27582.489,E2 27582.489} C_VEL
LIN {X 0,Y 220.484,Z 1202.737,A -85,B 0,C 180,E1 27583.258,E2 27583.258} C_VEL
LIN {X 0,Y 191.641,Z 1208.18,A -85,B 0,C 180,E1 27596.55,E2 27596.55} C_VEL
LIN {X 0,Y 179.099,Z 1208.094,A -85,B 0,C 180,E1 27610.323,E2 27610.323} C_VEL
LIN {X 0,Y 176.783,Z 1202.5,A -85,B 0,C 180,E1 27625.14,E2 27625.14} C_VEL
LIN {X 0,Y 177.42,Z 1196.777,A -85,B 0,C 180,E1 27632.483,E2 27632.483} C_VEL
LIN {X 0,Y 177.873,Z 1185.967,A -85,B 0,C 180,E1 27641.464,E2 27641.464} C_VEL
LIN {X 0,Y 179.029,Z 1176.915,A -85,B 0,C 180,E1 27647.226,E2 27647.226} C_VEL
LIN {X 0,Y 185.174,Z 1175.922,A -85,B 0,C 180,E1 27659.36,E2 27659.36} C_VEL
LIN {X 0,Y 200.408,Z 1168.977,A -85,B 0,C 180,E1 27669.905,E2 27669.905} C_VEL
LIN {X 0,Y 222.944,Z 1156.155,A -85,B 0,C 180,E1 27678.254,E2 27678.254} C_VEL
LIN {X 0,Y 247.826,Z 1138.923,A -85,B 0,C 180,E1 27683.937,E2 27683.937} C_VEL
LIN {X 0,Y 256.845,Z 1131.781,A -85,B 0,C 180,E1 27685.498,E2 27685.498} C_VEL
LIN {X 0,Y 256.516,Z 1131.988,A -85,B 0,C 180,E1 27686.033,E2 27686.033} C_VEL
LIN {X 0,Y 236.152,Z 1144.995,A -85,B 0,C 180,E1 27690.745,E2 27690.745} C_VEL
LIN {X 0,Y 219.966,Z 1151.621,A -85,B 0,C 180,E1 27695.663,E2 27695.663} C_VEL
LIN {X 0,Y 203.079,Z 1154.132,A -85,B 0,C 180,E1 27702.689,E2 27702.689} C_VEL
LIN {X 0,Y 190.138,Z 1150.844,A -85,B 0,C 180,E1 27710.859,E2 27710.859} C_VEL
LIN {X 0,Y 181.46,Z 1140.597,A -85,B 0,C 180,E1 27720.675,E2 27720.675} C_VEL
LIN {X 0,Y 178.528,Z 1125.146,A -85,B 0,C 180,E1 27729.751,E2 27729.751} C_VEL
LIN {X 0,Y 178.911,Z 1104.638,A -85,B 0,C 180,E1 27737.834,E2 27737.834} C_VEL
LIN {X 0,Y 180.769,Z 1080.63,A -85,B 0,C 180,E1 27744.343,E2 27744.343} C_VEL
LIN {X 0,Y 183.434,Z 1051.422,A -85,B 0,C 180,E1 27749.627,E2 27749.627} C_VEL
LIN {X 0,Y 185.8,Z 1019.533,A -85,B 0,C 180,E1 27753.152,E2 27753.152} C_VEL
LIN {X 0,Y 185.949,Z 993.549,A -85,B 0,C 180,E1 27754.906,E2 27754.906} C_VEL
LIN {X 0,Y 171.619,Z 923.03,A -85,B 0,C 180,E1 27760.454,E2 27760.454} C_VEL
LIN {X 0,Y 170.907,Z 923.03,A -85,B 0,C 180,E1 27770.887,E2 27770.887} C_VEL
LIN {X 0,Y 168.866,Z 923.03,A -85,B 0,C 180,E1 27775.226,E2 27775.226} C_VEL
LIN {X 0,Y 163.654,Z 923.03,A -85,B 0,C 180,E1 27782.695,E2 27782.695} C_VEL
LIN {X 0,Y 164.885,Z 923.03,A -85,B 0,C 180,E1 27793.995,E2 27793.995} C_VEL
LIN {X 0,Y 166.425,Z 923.03,A -85,B 0,C 180,E1 27804.745,E2 27804.745} C_VEL
LIN {X 0,Y 167.295,Z 923.03,A -85,B 0,C 180,E1 27809.954,E2 27809.954} C_VEL
LIN {X 0,Y 165.636,Z 923.03,A -85,B 0,C 180,E1 27820.465,E2 27820.465} C_VEL
LIN {X 0,Y 165.164,Z 923.131,A -85,B 0,C 180,E1 27824.016,E2 27824.016} C_VEL
LIN {X 0,Y 181.829,Z 962.414,A -85,B 0,C 180,E1 27833.365,E2 27833.365} C_VEL
LIN {X 0,Y 193.232,Z 997.744,A -85,B 0,C 180,E1 27840.505,E2 27840.505} C_VEL
LIN {X 0,Y 201.56,Z 1031.227,A -85,B 0,C 180,E1 27847.142,E2 27847.142} C_VEL
LIN {X 0,Y 205.741,Z 1053.359,A -85,B 0,C 180,E1 27851.682,E2 27851.682} C_VEL
LIN {X 0,Y 193.213,Z 1089.724,A -85,B 0,C 180,E1 27858.369,E2 27858.369} C_VEL
LIN {X 0,Y 181.984,Z 1121.342,A -85,B 0,C 180,E1 27866.844,E2 27866.844} C_VEL
LIN {X 0,Y 173.269,Z 1148.912,A -85,B 0,C 180,E1 27877.649,E2 27877.649} C_VEL
LIN {X 0,Y 169.115,Z 1169.29,A -85,B 0,C 180,E1 27889.115,E2 27889.115} C_VEL
LIN {X 0,Y 168.231,Z 1182.941,A -85,B 0,C 180,E1 27899.994,E2 27899.994} C_VEL
LIN {X 0,Y 170.851,Z 1194.192,A -85,B 0,C 180,E1 27913.584,E2 27913.584} C_VEL
LIN {X 0,Y 179.006,Z 1200.231,A -85,B 0,C 180,E1 27924.96,E2 27924.96} C_VEL
LIN {X 0,Y 198.487,Z 1203.555,A -85,B 0,C 180,E1 27937.515,E2 27937.515} C_VEL
LIN {X 0,Y 210.792,Z 1203.755,A -85,B 0,C 180,E1 27942.425,E2 27942.425} C_VEL
LIN {X 0,Y 208.97,Z 1204.236,A -85,B 0,C 180,E1 27943.746,E2 27943.746} C_VEL
LIN {X 0,Y 185.004,Z 1207.635,A -85,B 0,C 180,E1 27955.181,E2 27955.181} C_VEL
LIN {X 0,Y 171.625,Z 1207.007,A -85,B 0,C 180,E1 27969.428,E2 27969.428} C_VEL
LIN {X 0,Y 168.798,Z 1202.33,A -85,B 0,C 180,E1 27982.388,E2 27982.388} C_VEL
LIN {X 0,Y 169.684,Z 1196.111,A -85,B 0,C 180,E1 27991.321,E2 27991.321} C_VEL
LIN {X 0,Y 170.042,Z 1186.021,A -85,B 0,C 180,E1 28000.282,E2 28000.282} C_VEL
LIN {X 0,Y 171.51,Z 1174.98,A -85,B 0,C 180,E1 28008.006,E2 28008.006} C_VEL
LIN {X 0,Y 178.221,Z 1174.848,A -85,B 0,C 180,E1 28020.626,E2 28020.626} C_VEL
LIN {X 0,Y 194.343,Z 1168.881,A -85,B 0,C 180,E1 28031.417,E2 28031.417} C_VEL
LIN {X 0,Y 217.832,Z 1157.267,A -85,B 0,C 180,E1 28039.783,E2 28039.783} C_VEL
LIN {X 0,Y 243.241,Z 1141.575,A -85,B 0,C 180,E1 28045.324,E2 28045.324} C_VEL
LIN {X 0,Y 245.257,Z 1140.193,A -85,B 0,C 180,E1 28045.685,E2 28045.685} C_VEL
LIN {X 0,Y 244.765,Z 1140.382,A -85,B 0,C 180,E1 28046.25,E2 28046.25} C_VEL
LIN {X 0,Y 222.823,Z 1150.969,A -85,B 0,C 180,E1 28051.664,E2 28051.664} C_VEL
LIN {X 0,Y 203.708,Z 1155.318,A -85,B 0,C 180,E1 28058.234,E2 28058.234} C_VEL
LIN {X 0,Y 188.316,Z 1153.804,A -85,B 0,C 180,E1 28066.076,E2 28066.076} C_VEL
LIN {X 0,Y 177.373,Z 1146.445,A -85,B 0,C 180,E1 28075.118,E2 28075.118} C_VEL
LIN {X 0,Y 171.803,Z 1133.762,A -85,B 0,C 180,E1 28084.419,E2 28084.419} C_VEL
LIN {X 0,Y 170.63,Z 1115.606,A -85,B 0,C 180,E1 28093.35,E2 28093.35} C_VEL
LIN {X 0,Y 171.802,Z 1093.244,A -85,B 0,C 180,E1 28100.935,E2 28100.935} C_VEL
LIN {X 0,Y 174.303,Z 1064.733,A -85,B 0,C 180,E1 28107.429,E2 28107.429} C_VEL
LIN {X 0,Y 176.913,Z 1033.347,A -85,B 0,C 180,E1 28111.937,E2 28111.937} C_VEL
LIN {X 0,Y 178.437,Z 996.194,A -85,B 0,C 180,E1 28114.901,E2 28114.901} C_VEL
LIN {X 0,Y 163.657,Z 923.03,A -85,B 0,C 180,E1 28120.888,E2 28120.888} C_VEL
LIN {X 0,Y 162.747,Z 923.03,A -85,B 0,C 180,E1 28130.837,E2 28130.837} C_VEL
LIN {X 0,Y 163.211,Z 923.03,A -85,B 0,C 180,E1 28136.446,E2 28136.446} C_VEL
LIN {X 0,Y 163.654,Z 923.03,A -85,B 0,C 180,E1 28142.695,E2 28142.695} C_VEL
LIN {X 0,Y 161.449,Z 923.03,A -85,B 0,C 180,E1 28147.234,E2 28147.234} C_VEL
LIN {X 0,Y 157.002,Z 923.03,A -85,B 0,C 180,E1 28155.041,E2 28155.041} C_VEL
LIN {X 0,Y 158.412,Z 923.03,A -85,B 0,C 180,E1 28164.478,E2 28164.478} C_VEL
LIN {X 0,Y 159.372,Z 923.03,A -85,B 0,C 180,E1 28169.952,E2 28169.952} C_VEL
LIN {X 0,Y 157.581,Z 923.705,A -85,B 0,C 180,E1 28181.357,E2 28181.357} C_VEL
LIN {X 0,Y 173.543,Z 960.465,A -85,B 0,C 180,E1 28191.018,E2 28191.018} C_VEL
LIN {X 0,Y 184.778,Z 994.593,A -85,B 0,C 180,E1 28198.392,E2 28198.392} C_VEL
LIN {X 0,Y 193.677,Z 1030.119,A -85,B 0,C 180,E1 28205.762,E2 28205.762} C_VEL
LIN {X 0,Y 197.934,Z 1055.091,A -85,B 0,C 180,E1 28211.064,E2 28211.064} C_VEL
LIN {X 0,Y 184.762,Z 1092.17,A -85,B 0,C 180,E1 28218.234,E2 28218.234} C_VEL
LIN {X 0,Y 172.821,Z 1124.891,A -85,B 0,C 180,E1 28227.716,E2 28227.716} C_VEL
LIN {X 0,Y 164.888,Z 1150.387,A -85,B 0,C 180,E1 28238.489,E2 28238.489} C_VEL
LIN {X 0,Y 161.167,Z 1169.096,A -85,B 0,C 180,E1 28249.608,E2 28249.608} C_VEL
LIN {X 0,Y 160.468,Z 1183.134,A -85,B 0,C 180,E1 28261.343,E2 28261.343} C_VEL
LIN {X 0,Y 164.068,Z 1194.723,A -85,B 0,C 180,E1 28276.034,E2 28276.034} C_VEL
LIN {X 0,Y 177.533,Z 1201.858,A -85,B 0,C 180,E1 28290.704,E2 28290.704} C_VEL
LIN {X 0,Y 201.126,Z 1204.578,A -85,B 0,C 180,E1 28302.54,E2 28302.54} C_VEL
LIN {X 0,Y 172.463,Z 1207.129,A -85,B 0,C 180,E1 28318.339,E2 28318.339} C_VEL
LIN {X 0,Y 162.132,Z 1204.286,A -85,B 0,C 180,E1 28333.814,E2 28333.814} C_VEL
LIN {X 0,Y 161.618,Z 1197.467,A -85,B 0,C 180,E1 28347.368,E2 28347.368} C_VEL
LIN {X 0,Y 162.08,Z 1190.201,A -85,B 0,C 180,E1 28355.396,E2 28355.396} C_VEL
LIN {X 0,Y 163.163,Z 1175.827,A -85,B 0,C 180,E1 28366.178,E2 28366.178} C_VEL
LIN {X 0,Y 163.919,Z 1172.905,A -85,B 0,C 180,E1 28368.174,E2 28368.174} C_VEL
LIN {X 0,Y 167.17,Z 1174.16,A -85,B 0,C 180,E1 28376.918,E2 28376.918} C_VEL
LIN {X 0,Y 180.611,Z 1171.316,A -85,B 0,C 180,E1 28388.915,E2 28388.915} C_VEL
LIN {X 0,Y 202.377,Z 1163.059,A -85,B 0,C 180,E1 28398.354,E2 28398.354} C_VEL
LIN {X 0,Y 227.066,Z 1150.81,A -85,B 0,C 180,E1 28404.66,E2 28404.66} C_VEL
LIN {X 0,Y 233.695,Z 1146.924,A -85,B 0,C 180,E1 28406.284,E2 28406.284} C_VEL
LIN {X 0,Y 216.029,Z 1153.65,A -85,B 0,C 180,E1 28410.688,E2 28410.688} C_VEL
LIN {X 0,Y 196.367,Z 1156.788,A -85,B 0,C 180,E1 28417.376,E2 28417.376} C_VEL
LIN {X 0,Y 180.521,Z 1154.193,A -85,B 0,C 180,E1 28425.461,E2 28425.461} C_VEL
LIN {X 0,Y 169.36,Z 1145.738,A -85,B 0,C 180,E1 28434.887,E2 28434.887} C_VEL
LIN {X 0,Y 163.846,Z 1131.904,A -85,B 0,C 180,E1 28444.634,E2 28444.634} C_VEL
LIN {X 0,Y 162.847,Z 1113.825,A -85,B 0,C 180,E1 28453.459,E2 28453.459} C_VEL
LIN {X 0,Y 164.187,Z 1089.55,A -85,B 0,C 180,E1 28461.607,E2 28461.607} C_VEL
LIN {X 0,Y 166.728,Z 1061.113,A -85,B 0,C 180,E1 28467.966,E2 28467.966} C_VEL
LIN {X 0,Y 169.316,Z 1029.607,A -85,B 0,C 180,E1 28472.383,E2 28472.383} C_VEL
LIN {X 0,Y 170.237,Z 995.491,A -85,B 0,C 180,E1 28475.127,E2 28475.127} C_VEL
LIN {X 0,Y 155.683,Z 923.03,A -85,B 0,C 180,E1 28481.164,E2 28481.164} C_VEL
LIN {X 0,Y 154.941,Z 923.03,A -85,B 0,C 180,E1 28494.129,E2 28494.129} C_VEL
LIN {X 0,Y 155.491,Z 923.03,A -85,B 0,C 180,E1 28502.734,E2 28502.734} C_VEL
LIN {X 0,Y 156.768,Z 923.03,A -85,B 0,C 180,E1 28513.142,E2 28513.142} C_VEL
LIN {X 0,Y 157.002,Z 923.03,A -85,B 0,C 180,E1 28515.041,E2 28515.041} C_VEL
LIN {X 0,Y 154.887,Z 923.03,A -85,B 0,C 180,E1 28519.792,E2 28519.792} C_VEL
LIN {X 0,Y 150.929,Z 923.03,A -85,B 0,C 180,E1 28527.979,E2 28527.979} C_VEL
LIN {X 0,Y 151.15,Z 923.03,A -85,B 0,C 180,E1 28531.027,E2 28531.027} C_VEL
LIN {X 0,Y 149.944,Z 923.329,A -85,B 0,C 180,E1 28538.211,E2 28538.211} C_VEL
LIN {X 0,Y 164.836,Z 957.485,A -85,B 0,C 180,E1 28548.155,E2 28548.155} C_VEL
LIN {X 0,Y 175.849,Z 989.815,A -85,B 0,C 180,E1 28555.736,E2 28555.736} C_VEL
LIN {X 0,Y 184.864,Z 1025.141,A -85,B 0,C 180,E1 28563.434,E2 28563.434} C_VEL
LIN {X 0,Y 190.576,Z 1054.788,A -85,B 0,C 180,E1 28570.051,E2 28570.051} C_VEL
LIN {X 0,Y 177.744,Z 1090.502,A -85,B 0,C 180,E1 28577.14,E2 28577.14} C_VEL
LIN {X 0,Y 165.943,Z 1122.094,A -85,B 0,C 180,E1 28586.356,E2 28586.356} C_VEL
LIN {X 0,Y 157.463,Z 1148.035,A -85,B 0,C 180,E1 28597.421,E2 28597.421} C_VEL
LIN {X 0,Y 153.255,Z 1168.744,A -85,B 0,C 180,E1 28610.077,E2 28610.077} C_VEL
LIN {X 0,Y 152.661,Z 1181.882,A -85,B 0,C 180,E1 28621.412,E2 28621.412} C_VEL
LIN {X 0,Y 156.517,Z 1194.061,A -85,B 0,C 180,E1 28636.83,E2 28636.83} C_VEL
LIN {X 0,Y 170.763,Z 1201.865,A -85,B 0,C 180,E1 28652.063,E2 28652.063} C_VEL
LIN {X 0,Y 190.371,Z 1204.882,A -85,B 0,C 180,E1 28662.205,E2 28662.205} C_VEL
LIN {X 0,Y 188.471,Z 1205.313,A -85,B 0,C 180,E1 28663.878,E2 28663.878} C_VEL
LIN {X 0,Y 165.737,Z 1206.178,A -85,B 0,C 180,E1 28676.894,E2 28676.894} C_VEL
LIN {X 0,Y 154.592,Z 1202.845,A -85,B 0,C 180,E1 28693.001,E2 28693.001} C_VEL
LIN {X 0,Y 153.953,Z 1195.589,A -85,B 0,C 180,E1 28707.237,E2 28707.237} C_VEL
LIN {X 0,Y 154.373,Z 1188.054,A -85,B 0,C 180,E1 28715.667,E2 28715.667} C_VEL
LIN {X 0,Y 155.938,Z 1171.966,A -85,B 0,C 180,E1 28727.677,E2 28727.677} C_VEL
LIN {X 0,Y 156.46,Z 1170.783,A -85,B 0,C 180,E1 28729.073,E2 28729.073} C_VEL
LIN {X 0,Y 164.657,Z 1172.357,A -85,B 0,C 180,E1 28743.462,E2 28743.462} C_VEL
LIN {X 0,Y 182.673,Z 1168.282,A -85,B 0,C 180,E1 28754.732,E2 28754.732} C_VEL
LIN {X 0,Y 208.037,Z 1158.981,A -85,B 0,C 180,E1 28763.088,E2 28763.088} C_VEL
LIN {X 0,Y 220.788,Z 1153.155,A -85,B 0,C 180,E1 28765.938,E2 28765.938} C_VEL
LIN {X 0,Y 221.525,Z 1152.661,A -85,B 0,C 180,E1 28766.501,E2 28766.501} C_VEL
LIN {X 0,Y 198.777,Z 1157.767,A -85,B 0,C 180,E1 28772.868,E2 28772.868} C_VEL
LIN {X 0,Y 180.365,Z 1156.889,A -85,B 0,C 180,E1 28780.426,E2 28780.426} C_VEL
LIN {X 0,Y 166.372,Z 1150.206,A -85,B 0,C 180,E1 28789.54,E2 28789.54} C_VEL
LIN {X 0,Y 158.349,Z 1139.061,A -85,B 0,C 180,E1 28798.99,E2 28798.99} C_VEL
LIN {X 0,Y 155.162,Z 1121.753,A -85,B 0,C 180,E1 28809.112,E2 28809.112} C_VEL
LIN {X 0,Y 155.566,Z 1099.727,A -85,B 0,C 180,E1 28818.043,E2 28818.043} C_VEL
LIN {X 0,Y 157.689,Z 1073.502,A -85,B 0,C 180,E1 28825.286,E2 28825.286} C_VEL
LIN {X 0,Y 160.394,Z 1043.31,A -85,B 0,C 180,E1 28830.724,E2 28830.724} C_VEL
LIN {X 0,Y 162.578,Z 1009.785,A -85,B 0,C 180,E1 28834.184,E2 28834.184} C_VEL
LIN {X 0,Y 162.059,Z 994.81,A -85,B 0,C 180,E1 28835.33,E2 28835.33} C_VEL
LIN {X 0,Y 147.622,Z 923.03,A -85,B 0,C 180,E1 28841.919,E2 28841.919} C_VEL
LIN {X 0,Y 146.981,Z 923.03,A -85,B 0,C 180,E1 28855.344,E2 28855.344} C_VEL
LIN {X 0,Y 148.102,Z 923.03,A -85,B 0,C 180,E1 28866.691,E2 28866.691} C_VEL
LIN {X 0,Y 149.488,Z 923.03,A -85,B 0,C 180,E1 28878.285,E2 28878.285} C_VEL
LIN {X 0,Y 150.929,Z 923.03,A -85,B 0,C 180,E1 28887.979,E2 28887.979} C_VEL
LIN {X 0,Y 148.563,Z 923.03,A -85,B 0,C 180,E1 28889.877,E2 28889.877} C_VEL
LIN {X 0,Y 142.811,Z 923.03,A -85,B 0,C 180,E1 28892.994,E2 28892.994} C_VEL
LIN {X 0,Y 142.623,Z 923.652,A -85,B 0,C 180,E1 28894.884,E2 28894.884} C_VEL
LIN {X 0,Y 156.194,Z 954.521,A -85,B 0,C 180,E1 28904.969,E2 28904.969} C_VEL
LIN {X 0,Y 166.682,Z 984.065,A -85,B 0,C 180,E1 28912.61,E2 28912.61} C_VEL
LIN {X 0,Y 175.881,Z 1018.68,A -85,B 0,C 180,E1 28920.619,E2 28920.619} C_VEL
LIN {X 0,Y 182.325,Z 1051.933,A -85,B 0,C 180,E1 28928.302,E2 28928.302} C_VEL
LIN {X 0,Y 182.537,Z 1057.759,A -85,B 0,C 180,E1 28929.613,E2 28929.613} C_VEL
LIN {X 0,Y 168.242,Z 1095.445,A -85,B 0,C 180,E1 28937.645,E2 28937.645} C_VEL
LIN {X 0,Y 156.241,Z 1126.905,A -85,B 0,C 180,E1 28947.857,E2 28947.857} C_VEL
LIN {X 0,Y 148.719,Z 1150.825,A -85,B 0,C 180,E1 28959.161,E2 28959.161} C_VEL
LIN {X 0,Y 145.299,Z 1168.719,A -85,B 0,C 180,E1 28970.909,E2 28970.909} C_VEL
LIN {X 0,Y 144.922,Z 1181.954,A -85,B 0,C 180,E1 28982.982,E2 28982.982} C_VEL
LIN {X 0,Y 149.001,Z 1193.317,A -85,B 0,C 180,E1 28997.706,E2 28997.706} C_VEL
LIN {X 0,Y 164.091,Z 1201.645,A -85,B 0,C 180,E1 29013.534,E2 29013.534} C_VEL
LIN {X 0,Y 180.239,Z 1204.763,A -85,B 0,C 180,E1 29022.115,E2 29022.115} C_VEL
LIN {X 0,Y 180.671,Z 1204.974,A -85,B 0,C 180,E1 29023.024,E2 29023.024} C_VEL
LIN {X 0,Y 159.118,Z 1205.117,A -85,B 0,C 180,E1 29035.325,E2 29035.325} C_VEL
LIN {X 0,Y 147.095,Z 1201.266,A -85,B 0,C 180,E1 29052.106,E2 29052.106} C_VEL
LIN {X 0,Y 146.327,Z 1193.597,A -85,B 0,C 180,E1 29067.093,E2 29067.093} C_VEL
LIN {X 0,Y 146.698,Z 1185.711,A -85,B 0,C 180,E1 29075.964,E2 29075.964} C_VEL
LIN {X 0,Y 149.002,Z 1168.246,A -85,B 0,C 180,E1 29089.297,E2 29089.297} C_VEL
LIN {X 0,Y 153.22,Z 1170.666,A -85,B 0,C 180,E1 29099.6,E2 29099.6} C_VEL
LIN {X 0,Y 164.661,Z 1170.219,A -85,B 0,C 180,E1 29110.026,E2 29110.026} C_VEL
LIN {X 0,Y 186.923,Z 1165.047,A -85,B 0,C 180,E1 29120.231,E2 29120.231} C_VEL
LIN {X 0,Y 209.288,Z 1157.281,A -85,B 0,C 180,E1 29126.189,E2 29126.189} C_VEL
LIN {X 0,Y 208.913,Z 1157.149,A -85,B 0,C 180,E1 29126.837,E2 29126.837} C_VEL
LIN {X 0,Y 184.52,Z 1159.33,A -85,B 0,C 180,E1 29134.351,E2 29134.351} C_VEL
LIN {X 0,Y 168.763,Z 1155.955,A -85,B 0,C 180,E1 29141.742,E2 29141.742} C_VEL
LIN {X 0,Y 155.757,Z 1146.824,A -85,B 0,C 180,E1 29151.638,E2 29151.638} C_VEL
LIN {X 0,Y 148.651,Z 1131.13,A -85,B 0,C 180,E1 29162.92,E2 29162.92} C_VEL
LIN {X 0,Y 147.329,Z 1112.063,A -85,B 0,C 180,E1 29172.65,E2 29172.65} C_VEL
LIN {X 0,Y 148.547,Z 1087.691,A -85,B 0,C 180,E1 29181.254,E2 29181.254} C_VEL
LIN {X 0,Y 151.07,Z 1059.335,A -85,B 0,C 180,E1 29187.974,E2 29187.974} C_VEL
LIN {X 0,Y 153.617,Z 1027.999,A -85,B 0,C 180,E1 29192.589,E2 29192.589} C_VEL
LIN {X 0,Y 154.666,Z 998.006,A -85,B 0,C 180,E1 29195.208,E2 29195.208} C_VEL
LIN {X 0,Y 139.648,Z 923.03,A -85,B 0,C 180,E1 29202.277,E2 29202.277} C_VEL
LIN {X 0,Y 139.109,Z 923.03,A -85,B 0,C 180,E1 29217.041,E2 29217.041} C_VEL
LIN {X 0,Y 139.667,Z 923.03,A -85,B 0,C 180,E1 29224.298,E2 29224.298} C_VEL
LIN {X 0,Y 140.894,Z 923.03,A -85,B 0,C 180,E1 29234.877,E2 29234.877} C_VEL
LIN {X 0,Y 142.365,Z 923.03,A -85,B 0,C 180,E1 29243.854,E2 29243.854} C_VEL
LIN {X 0,Y 143.499,Z 923.03,A -85,B 0,C 180,E1 29249.947,E2 29249.947} C_VEL
LIN {X 0,Y 142.811,Z 923.03,A -85,B 0,C 180,E1 29252.994,E2 29252.994} C_VEL
LIN {X 0,Y 143.452,Z 925.882,A -85,B 0,C 180,E1 29255.537,E2 29255.537} C_VEL
LIN {X 0,Y 145.208,Z 933.773,A -85,B 0,C 180,E1 29257.712,E2 29257.712} C_VEL
LIN {X 0,Y 147.482,Z 950.98,A -85,B 0,C 180,E1 29261.264,E2 29261.264} C_VEL
LIN {X 0,Y 158.292,Z 980.713,A -85,B 0,C 180,E1 29269.725,E2 29269.725} C_VEL
LIN {X 0,Y 167.453,Z 1015.116,A -85,B 0,C 180,E1 29278.224,E2 29278.224} C_VEL
LIN {X 0,Y 174.239,Z 1049.416,A -85,B 0,C 180,E1 29286.543,E2 29286.543} C_VEL
LIN {X 0,Y 175.084,Z 1058.337,A -85,B 0,C 180,E1 29288.694,E2 29288.694} C_VEL
LIN {X 0,Y 160.488,Z 1095.632,A -85,B 0,C 180,E1 29296.942,E2 29296.942} C_VEL
LIN {X 0,Y 148.203,Z 1127.026,A -85,B 0,C 180,E1 29307.629,E2 29307.629} C_VEL
LIN {X 0,Y 140.617,Z 1150.915,A -85,B 0,C 180,E1 29319.552,E2 29319.552} C_VEL
LIN {X 0,Y 137.364,Z 1168.847,A -85,B 0,C 180,E1 29332.033,E2 29332.033} C_VEL
LIN {X 0,Y 137.264,Z 1181.952,A -85,B 0,C 180,E1 29344.729,E2 29344.729} C_VEL
LIN {X 0,Y 143.295,Z 1194.258,A -85,B 0,C 180,E1 29361.652,E2 29361.652} C_VEL
LIN {X 0,Y 165.485,Z 1203.385,A -85,B 0,C 180,E1 29379.724,E2 29379.724} C_VEL
LIN {X 0,Y 170.34,Z 1204.244,A -85,B 0,C 180,E1 29382.064,E2 29382.064} C_VEL
LIN {X 0,Y 170.106,Z 1204.496,A -85,B 0,C 180,E1 29383.334,E2 29383.334} C_VEL
LIN {X 0,Y 146.821,Z 1203.045,A -85,B 0,C 180,E1 29399.093,E2 29399.093} C_VEL
LIN {X 0,Y 138.371,Z 1196.929,A -85,B 0,C 180,E1 29417.442,E2 29417.442} C_VEL
LIN {X 0,Y 139.093,Z 1189.197,A -85,B 0,C 180,E1 29430.055,E2 29430.055} C_VEL
LIN {X 0,Y 139.259,Z 1177.241,A -85,B 0,C 180,E1 29441.532,E2 29441.532} C_VEL
LIN {X 0,Y 141.744,Z 1165.763,A -85,B 0,C 180,E1 29450.327,E2 29450.327} C_VEL
LIN {X 0,Y 151.671,Z 1169.186,A -85,B 0,C 180,E1 29466.77,E2 29466.77} C_VEL
LIN {X 0,Y 167.025,Z 1167.788,A -85,B 0,C 180,E1 29476.427,E2 29476.427} C_VEL
LIN {X 0,Y 192.497,Z 1161.847,A -85,B 0,C 180,E1 29485.178,E2 29485.178} C_VEL
LIN {X 0,Y 197.282,Z 1160.199,A -85,B 0,C 180,E1 29486.918,E2 29486.918} C_VEL
LIN {X 0,Y 174.476,Z 1159.862,A -85,B 0,C 180,E1 29494.345,E2 29494.345} C_VEL
LIN {X 0,Y 157.26,Z 1153.8,A -85,B 0,C 180,E1 29503.252,E2 29503.252} C_VEL
LIN {X 0,Y 145.44,Z 1142.059,A -85,B 0,C 180,E1 29514.043,E2 29514.043} C_VEL
LIN {X 0,Y 140.149,Z 1124.585,A -85,B 0,C 180,E1 29525.42,E2 29525.42} C_VEL
LIN {X 0,Y 139.749,Z 1103.201,A -85,B 0,C 180,E1 29535.369,E2 29535.369} C_VEL
LIN {X 0,Y 141.528,Z 1077.395,A -85,B 0,C 180,E1 29543.61,E2 29543.61} C_VEL
LIN {X 0,Y 144.224,Z 1047.59,A -85,B 0,C 180,E1 29549.854,E2 29549.854} C_VEL
LIN {X 0,Y 146.569,Z 1015.065,A -85,B 0,C 180,E1 29553.857,E2 29553.857} C_VEL
LIN {X 0,Y 146.231,Z 996.184,A -85,B 0,C 180,E1 29555.471,E2 29555.471} C_VEL
LIN {X 0,Y 131.633,Z 923.03,A -85,B 0,C 180,E1 29562.868,E2 29562.868} C_VEL
LIN {X 0,Y 130.886,Z 923.03,A -85,B 0,C 180,E1 29574.675,E2 29574.675} C_VEL
LIN {X 0,Y 131.818,Z 923.03,A -85,B 0,C 180,E1 29586.521,E2 29586.521} C_VEL
LIN {X 0,Y 133.281,Z 923.03,A -85,B 0,C 180,E1 29596.836,E2 29596.836} C_VEL
LIN {X 0,Y 135.556,Z 923.03,A -85,B 0,C 180,E1 29609.944,E2 29609.944} C_VEL
LIN {X 0,Y 135.331,Z 923.742,A -85,B 0,C 180,E1 29611.022,E2 29611.022} C_VEL
LIN {X 0,Y 147.482,Z 950.98,A -85,B 0,C 180,E1 29621.264,E2 29621.264} C_VEL
LIN {X 0,Y 149.706,Z 962.079,A -85,B 0,C 180,E1 29623.821,E2 29623.821} C_VEL
LIN {X 0,Y 151.368,Z 981.629,A -85,B 0,C 180,E1 29627.757,E2 29627.757} C_VEL
LIN {X 0,Y 160.327,Z 1016.601,A -85,B 0,C 180,E1 29636.918,E2 29636.918} C_VEL
LIN {X 0,Y 166.737,Z 1050.236,A -85,B 0,C 180,E1 29645.503,E2 29645.503} C_VEL
LIN {X 0,Y 167.397,Z 1059.492,A -85,B 0,C 180,E1 29647.82,E2 29647.82} C_VEL
LIN {X 0,Y 152.231,Z 1097.005,A -85,B 0,C 180,E1 29656.57,E2 29656.57} C_VEL
LIN {X 0,Y 140.182,Z 1127.052,A -85,B 0,C 180,E1 29667.378,E2 29667.378} C_VEL
LIN {X 0,Y 132.527,Z 1150.92,A -85,B 0,C 180,E1 29679.99,E2 29679.99} C_VEL
LIN {X 0,Y 129.469,Z 1168.876,A -85,B 0,C 180,E1 29693.29,E2 29693.29} C_VEL
LIN {X 0,Y 129.734,Z 1181.884,A -85,B 0,C 180,E1 29706.682,E2 29706.682} C_VEL
LIN {X 0,Y 138.363,Z 1195.104,A -85,B 0,C 180,E1 29725.896,E2 29725.896} C_VEL
LIN {X 0,Y 160.791,Z 1203.399,A -85,B 0,C 180,E1 29742.176,E2 29742.176} C_VEL
LIN {X 0,Y 157.889,Z 1203.497,A -85,B 0,C 180,E1 29744.56,E2 29744.56} C_VEL
LIN {X 0,Y 135.378,Z 1199.946,A -85,B 0,C 180,E1 29763.547,E2 29763.547} C_VEL
LIN {X 0,Y 130.62,Z 1192.652,A -85,B 0,C 180,E1 29781.279,E2 29781.279} C_VEL
LIN {X 0,Y 131.403,Z 1185.536,A -85,B 0,C 180,E1 29791.705,E2 29791.705} C_VEL
LIN {X 0,Y 131.888,Z 1171.994,A -85,B 0,C 180,E1 29804.15,E2 29804.15} C_VEL
LIN {X 0,Y 134.542,Z 1162.948,A -85,B 0,C 180,E1 29811.036,E2 29811.036} C_VEL
LIN {X 0,Y 139.805,Z 1166.564,A -85,B 0,C 180,E1 29822.774,E2 29822.774} C_VEL
LIN {X 0,Y 152.847,Z 1167.403,A -85,B 0,C 180,E1 29833.856,E2 29833.856} C_VEL
LIN {X 0,Y 177.171,Z 1164.202,A -85,B 0,C 180,E1 29844.187,E2 29844.187} C_VEL
LIN {X 0,Y 184.389,Z 1162.65,A -85,B 0,C 180,E1 29846.224,E2 29846.224} C_VEL
LIN {X 0,Y 185.625,Z 1162.159,A -85,B 0,C 180,E1 29846.996,E2 29846.996} C_VEL
LIN {X 0,Y 167.263,Z 1160.412,A -85,B 0,C 180,E1 29853.153,E2 29853.153} C_VEL
LIN {X 0,Y 149.549,Z 1153.188,A -85,B 0,C 180,E1 29862.361,E2 29862.361} C_VEL
LIN {X 0,Y 137.539,Z 1140.247,A -85,B 0,C 180,E1 29873.699,E2 29873.699} C_VEL
LIN {X 0,Y 132.339,Z 1121.49,A -85,B 0,C 180,E1 29885.741,E2 29885.741} C_VEL
LIN {X 0,Y 132.156,Z 1098.721,A -85,B 0,C 180,E1 29896.19,E2 29896.19} C_VEL
LIN {X 0,Y 134.127,Z 1071.377,A -85,B 0,C 180,E1 29904.669,E2 29904.669} C_VEL
LIN {X 0,Y 136.846,Z 1041.001,A -85,B 0,C 180,E1 29910.719,E2 29910.719} C_VEL
LIN {X 0,Y 139.134,Z 1004.504,A -85,B 0,C 180,E1 29914.798,E2 29914.798} C_VEL
LIN {X 0,Y 123.643,Z 923.03,A -85,B 0,C 180,E1 29923.426,E2 29923.426} C_VEL
LIN {X 0,Y 123.201,Z 923.03,A -85,B 0,C 180,E1 29940.551,E2 29940.551} C_VEL
LIN {X 0,Y 124.122,Z 923.03,A -85,B 0,C 180,E1 29948.515,E2 29948.515} C_VEL
LIN {X 0,Y 125.1,Z 923.03,A -85,B 0,C 180,E1 29955.959,E2 29955.959} C_VEL
LIN {X 0,Y 126.641,Z 923.65,A -85,B 0,C 180,E1 29965.449,E2 29965.449} C_VEL
LIN {X 0,Y 129.806,Z 928.851,A -85,B 0,C 180,E1 29968.691,E2 29968.691} C_VEL
LIN {X 0,Y 136.938,Z 943.63,A -85,B 0,C 180,E1 29975.405,E2 29975.405} C_VEL
LIN {X 0,Y 146.511,Z 967.277,A -85,B 0,C 180,E1 29983.554,E2 29983.554} C_VEL
LIN {X 0,Y 151.368,Z 981.629,A -85,B 0,C 180,E1 29987.757,E2 29987.757} C_VEL
LIN {X 0,Y 152.371,Z 993.01,A -85,B 0,C 180,E1 29990.187,E2 29990.187} C_VEL
LIN {X 0,Y 152.054,Z 1012.587,A -85,B 0,C 180,E1 29994.068,E2 29994.068} C_VEL
LIN {X 0,Y 158.296,Z 1045.207,A -85,B 0,C 180,E1 30002.821,E2 30002.821} C_VEL
LIN {X 0,Y 160.084,Z 1059.665,A -85,B 0,C 180,E1 30006.72,E2 30006.72} C_VEL
LIN {X 0,Y 144.539,Z 1096.968,A -85,B 0,C 180,E1 30015.742,E2 30015.742} C_VEL
LIN {X 0,Y 132.191,Z 1127.011,A -85,B 0,C 180,E1 30027.105,E2 30027.105} C_VEL
LIN {X 0,Y 124.467,Z 1150.86,A -85,B 0,C 180,E1 30040.489,E2 30040.489} C_VEL
LIN {X 0,Y 121.65,Z 1169.018,A -85,B 0,C 180,E1 30054.893,E2 30054.893} C_VEL
LIN {X 0,Y 122.056,Z 1180.293,A -85,B 0,C 180,E1 30067.104,E2 30067.104} C_VEL
LIN {X 0,Y 128.822,Z 1192.193,A -85,B 0,C 180,E1 30084.232,E2 30084.232} C_VEL
LIN {X 0,Y 150.618,Z 1202.011,A -85,B 0,C 180,E1 30101.985,E2 30101.985} C_VEL
LIN {X 0,Y 151.137,Z 1202.321,A -85,B 0,C 180,E1 30103.088,E2 30103.088} C_VEL
LIN {X 0,Y 126.447,Z 1197.084,A -85,B 0,C 180,E1 30125.507,E2 30125.507} C_VEL
LIN {X 0,Y 123.352,Z 1188.159,A -85,B 0,C 180,E1 30144.791,E2 30144.791} C_VEL
LIN {X 0,Y 123.808,Z 1181.493,A -85,B 0,C 180,E1 30153.56,E2 30153.56} C_VEL
LIN {X 0,Y 125.07,Z 1165.598,A -85,B 0,C 180,E1 30167.643,E2 30167.643} C_VEL
LIN {X 0,Y 127.454,Z 1159.933,A -85,B 0,C 180,E1 30171.809,E2 30171.809} C_VEL
LIN {X 0,Y 133.352,Z 1164.266,A -85,B 0,C 180,E1 30184.578,E2 30184.578} C_VEL
LIN {X 0,Y 147.261,Z 1165.728,A -85,B 0,C 180,E1 30195.983,E2 30195.983} C_VEL
LIN {X 0,Y 173.137,Z 1163.386,A -85,B 0,C 180,E1 30206.457,E2 30206.457} C_VEL
LIN {X 0,Y 172.961,Z 1163.022,A -85,B 0,C 180,E1 30207.314,E2 30207.314} C_VEL
LIN {X 0,Y 155.113,Z 1159.139,A -85,B 0,C 180,E1 30214.006,E2 30214.006} C_VEL
LIN {X 0,Y 138.287,Z 1149.41,A -85,B 0,C 180,E1 30224.153,E2 30224.153} C_VEL
LIN {X 0,Y 127.649,Z 1133.519,A -85,B 0,C 180,E1 30236.614,E2 30236.614} C_VEL
LIN {X 0,Y 124.369,Z 1113.405,A -85,B 0,C 180,E1 30248.525,E2 30248.525} C_VEL
LIN {X 0,Y 124.882,Z 1089.703,A -85,B 0,C 180,E1 30258.528,E2 30258.528} C_VEL
LIN {X 0,Y 127.074,Z 1062.178,A -85,B 0,C 180,E1 30266.392,E2 30266.392} C_VEL
LIN {X 0,Y 129.665,Z 1030.941,A -85,B 0,C 180,E1 30271.984,E2 30271.984} C_VEL
LIN {X 0,Y 130.86,Z 999.734,A -85,B 0,C 180,E1 30275.275,E2 30275.275} C_VEL
LIN {X 0,Y 115.642,Z 923.03,A -85,B 0,C 180,E1 30283.925,E2 30283.925} C_VEL
LIN {X 0,Y 115,Z 923.03,A -85,B 0,C 180,E1 30298.217,E2 30298.217} C_VEL
LIN {X 0,Y 115.803,Z 923.03,A -85,B 0,C 180,E1 30306.885,E2 30306.885} C_VEL
LIN {X 0,Y 117.346,Z 923.686,A -85,B 0,C 180,E1 30317.62,E2 30317.62} C_VEL
LIN {X 0,Y 120.672,Z 928.906,A -85,B 0,C 180,E1 30322.065,E2 30322.065} C_VEL
LIN {X 0,Y 123.173,Z 931.511,A -85,B 0,C 180,E1 30324.692,E2 30324.692} C_VEL
LIN {X 0,Y 127.824,Z 939.039,A -85,B 0,C 180,E1 30329.493,E2 30329.493} C_VEL
LIN {X 0,Y 137.788,Z 962.631,A -85,B 0,C 180,E1 30339.201,E2 30339.201} C_VEL
LIN {X 0,Y 146.623,Z 990.588,A -85,B 0,C 180,E1 30347.953,E2 30347.953} C_VEL
LIN {X 0,Y 152.054,Z 1012.587,A -85,B 0,C 180,E1 30354.068,E2 30354.068} C_VEL
LIN {X 0,Y 152.412,Z 1020.096,A -85,B 0,C 180,E1 30355.765,E2 30355.765} C_VEL
LIN {X 0,Y 150.165,Z 1041.315,A -85,B 0,C 180,E1 30360.204,E2 30360.204} C_VEL
LIN {X 0,Y 150.364,Z 1043.08,A -85,B 0,C 180,E1 30360.705,E2 30360.705} C_VEL
LIN {X 0,Y 152.23,Z 1061.141,A -85,B 0,C 180,E1 30365.783,E2 30365.783} C_VEL
LIN {X 0,Y 136.249,Z 1098.427,A -85,B 0,C 180,E1 30375.353,E2 30375.353} C_VEL
LIN {X 0,Y 123.538,Z 1128.552,A -85,B 0,C 180,E1 30387.638,E2 30387.638} C_VEL
LIN {X 0,Y 116.047,Z 1151.948,A -85,B 0,C 180,E1 30401.977,E2 30401.977} C_VEL
LIN {X 0,Y 113.907,Z 1168.249,A -85,B 0,C 180,E1 30415.91,E2 30415.91} C_VEL
LIN {X 0,Y 114.822,Z 1180.48,A -85,B 0,C 180,E1 30430.082,E2 30430.082} C_VEL
LIN {X 0,Y 124.441,Z 1192.958,A -85,B 0,C 180,E1 30449.051,E2 30449.051} C_VEL
LIN {X 0,Y 140.704,Z 1200.221,A -85,B 0,C 180,E1 30461.849,E2 30461.849} C_VEL
LIN {X 0,Y 141.289,Z 1200.572,A -85,B 0,C 180,E1 30463.204,E2 30463.204} C_VEL
LIN {X 0,Y 119.427,Z 1195.036,A -85,B 0,C 180,E1 30483.994,E2 30483.994} C_VEL
LIN {X 0,Y 115.841,Z 1185.82,A -85,B 0,C 180,E1 30504.452,E2 30504.452} C_VEL
LIN {X 0,Y 116.209,Z 1178.835,A -85,B 0,C 180,E1 30513.793,E2 30513.793} C_VEL
LIN {X 0,Y 119.907,Z 1157.706,A -85,B 0,C 180,E1 30532.28,E2 30532.28} C_VEL
LIN {X 0,Y 120.727,Z 1157.384,A -85,B 0,C 180,E1 30534.07,E2 30534.07} C_VEL
LIN {X 0,Y 127.086,Z 1161.804,A -85,B 0,C 180,E1 30546.549,E2 30546.549} C_VEL
LIN {X 0,Y 141.938,Z 1163.888,A -85,B 0,C 180,E1 30558.254,E2 30558.254} C_VEL
LIN {X 0,Y 162.577,Z 1163.146,A -85,B 0,C 180,E1 30566.852,E2 30566.852} C_VEL
LIN {X 0,Y 140.787,Z 1155.399,A -85,B 0,C 180,E1 30576.225,E2 30576.225} C_VEL
LIN {X 0,Y 125.755,Z 1142.414,A -85,B 0,C 180,E1 30587.793,E2 30587.793} C_VEL
LIN {X 0,Y 118.079,Z 1123.782,A -85,B 0,C 180,E1 30600.924,E2 30600.924} C_VEL
LIN {X 0,Y 116.712,Z 1101.228,A -85,B 0,C 180,E1 30612.852,E2 30612.852} C_VEL
LIN {X 0,Y 118.2,Z 1074.472,A -85,B 0,C 180,E1 30622.561,E2 30622.561} C_VEL
LIN {X 0,Y 120.758,Z 1044.308,A -85,B 0,C 180,E1 30629.643,E2 30629.643} C_VEL
LIN {X 0,Y 123.152,Z 1008.164,A -85,B 0,C 180,E1 30634.388,E2 30634.388} C_VEL
LIN {X 0,Y 121.729,Z 994.517,A -85,B 0,C 180,E1 30635.798,E2 30635.798} C_VEL
LIN {X 0,Y 107.609,Z 923.03,A -85,B 0,C 180,E1 30644.61,E2 30644.61} C_VEL
LIN {X 0,Y 107.122,Z 923.03,A -85,B 0,C 180,E1 30661.457,E2 30661.457} C_VEL
LIN {X 0,Y 107.648,Z 924.294,A -85,B 0,C 180,E1 30665.019,E2 30665.019} C_VEL
LIN {X 0,Y 112.526,Z 929.716,A -85,B 0,C 180,E1 30674.352,E2 30674.352} C_VEL
LIN {X 0,Y 114.358,Z 931.859,A -85,B 0,C 180,E1 30677.025,E2 30677.025} C_VEL
LIN {X 0,Y 120.109,Z 939.205,A -85,B 0,C 180,E1 30684.154,E2 30684.154} C_VEL
LIN {X 0,Y 124.797,Z 947.206,A -85,B 0,C 180,E1 30689.251,E2 30689.251} C_VEL
LIN {X 0,Y 133.445,Z 970.253,A -85,B 0,C 180,E1 30698.736,E2 30698.736} C_VEL
LIN {X 0,Y 141.459,Z 998.143,A -85,B 0,C 180,E1 30707.827,E2 30707.827} C_VEL
LIN {X 0,Y 148.424,Z 1031.21,A -85,B 0,C 180,E1 30717.351,E2 30717.351} C_VEL
LIN {X 0,Y 150.364,Z 1043.08,A -85,B 0,C 180,E1 30720.705,E2 30720.705} C_VEL
LIN {X 0,Y 149.508,Z 1052.419,A -85,B 0,C 180,E1 30722.927,E2 30722.927} C_VEL
LIN {X 0,Y 139.926,Z 1072.889,A -85,B 0,C 180,E1 30727.098,E2 30727.098} C_VEL
LIN {X 0,Y 123.953,Z 1108.496,A -85,B 0,C 180,E1 30738.152,E2 30738.152} C_VEL
LIN {X 0,Y 112.415,Z 1137.003,A -85,B 0,C 180,E1 30752.373,E2 30752.373} C_VEL
LIN {X 0,Y 106.721,Z 1160.043,A -85,B 0,C 180,E1 30769.797,E2 30769.797} C_VEL
LIN {X 0,Y 106.397,Z 1173.535,A -85,B 0,C 180,E1 30784.052,E2 30784.052} C_VEL
LIN {X 0,Y 112.381,Z 1187.397,A -85,B 0,C 180,E1 30803.781,E2 30803.781} C_VEL
LIN {X 0,Y 131.428,Z 1198.157,A -85,B 0,C 180,E1 30822.057,E2 30822.057} C_VEL
LIN {X 0,Y 131.278,Z 1198.377,A -85,B 0,C 180,E1 30823.557,E2 30823.557} C_VEL
LIN {X 0,Y 110.836,Z 1191.654,A -85,B 0,C 180,E1 30845.935,E2 30845.935} C_VEL
LIN {X 0,Y 108.664,Z 1182.111,A -85,B 0,C 180,E1 30866.084,E2 30866.084} C_VEL
LIN {X 0,Y 108.61,Z 1174.242,A -85,B 0,C 180,E1 30876.06,E2 30876.06} C_VEL
LIN {X 0,Y 113.178,Z 1154.351,A -85,B 0,C 180,E1 30893.684,E2 30893.684} C_VEL
LIN {X 0,Y 113.982,Z 1154.19,A -85,B 0,C 180,E1 30895.547,E2 30895.547} C_VEL
LIN {X 0,Y 127.358,Z 1160.682,A -85,B 0,C 180,E1 30914.621,E2 30914.621} C_VEL
LIN {X 0,Y 148.883,Z 1162.135,A -85,B 0,C 180,E1 30926.033,E2 30926.033} C_VEL
LIN {X 0,Y 150.304,Z 1161.825,A -85,B 0,C 180,E1 30927.219,E2 30927.219} C_VEL
LIN {X 0,Y 128.738,Z 1151.219,A -85,B 0,C 180,E1 30937.741,E2 30937.741} C_VEL
LIN {X 0,Y 114.951,Z 1134.845,A -85,B 0,C 180,E1 30951.031,E2 30951.031} C_VEL
LIN {X 0,Y 109.545,Z 1113.513,A -85,B 0,C 180,E1 30964.954,E2 30964.954} C_VEL
LIN {X 0,Y 109.362,Z 1090.333,A -85,B 0,C 180,E1 30976.051,E2 30976.051} C_VEL
LIN {X 0,Y 111.371,Z 1061.69,A -85,B 0,C 180,E1 30985.337,E2 30985.337} C_VEL
LIN {X 0,Y 113.857,Z 1030.629,A -85,B 0,C 180,E1 30991.524,E2 30991.524} C_VEL
LIN {X 0,Y 114.854,Z 1000.32,A -85,B 0,C 180,E1 30995.155,E2 30995.155} C_VEL
LIN {X 0,Y 101.074,Z 930.343,A -85,B 0,C 180,E1 31004.271,E2 31004.271} C_VEL
LIN {X 0,Y 101.527,Z 928.553,A -85,B 0,C 180,E1 31006.772,E2 31006.772} C_VEL
LIN {X 0,Y 105.001,Z 931.318,A -85,B 0,C 180,E1 31023.691,E2 31023.691} C_VEL
LIN {X 0,Y 110.307,Z 937.3,A -85,B 0,C 180,E1 31034.321,E2 31034.321} C_VEL
LIN {X 0,Y 117.545,Z 947.287,A -85,B 0,C 180,E1 31044.109,E2 31044.109} C_VEL
LIN {X 0,Y 122.506,Z 958.601,A -85,B 0,C 180,E1 31050.319,E2 31050.319} C_VEL
LIN {X 0,Y 129.975,Z 981.21,A -85,B 0,C 180,E1 31059.56,E2 31059.56} C_VEL
LIN {X 0,Y 136.869,Z 1009.395,A -85,B 0,C 180,E1 31068.863,E2 31068.863} C_VEL
LIN {X 0,Y 142.742,Z 1042.331,A -85,B 0,C 180,E1 31078.817,E2 31078.817} C_VEL
LIN {X 0,Y 144.913,Z 1061.436,A -85,B 0,C 180,E1 31084.545,E2 31084.545} C_VEL
LIN {X 0,Y 139.926,Z 1072.889,A -85,B 0,C 180,E1 31087.098,E2 31087.098} C_VEL
LIN {X 0,Y 130.317,Z 1086.001,A -85,B 0,C 180,E1 31089.916,E2 31089.916} C_VEL
LIN {X 0,Y 120.753,Z 1098.496,A -85,B 0,C 180,E1 31093.503,E2 31093.503} C_VEL
LIN {X 0,Y 107.7,Z 1127.679,A -85,B 0,C 180,E1 31106.844,E2 31106.844} C_VEL
LIN {X 0,Y 100.104,Z 1151.427,A -85,B 0,C 180,E1 31123.549,E2 31123.549} C_VEL
LIN {X 0,Y 98.537,Z 1167.842,A -85,B 0,C 180,E1 31139.991,E2 31139.991} C_VEL
LIN {X 0,Y 102.248,Z 1181.985,A -85,B 0,C 180,E1 31159.412,E2 31159.412} C_VEL
LIN {X 0,Y 121.831,Z 1195.598,A -85,B 0,C 180,E1 31182.01,E2 31182.01} C_VEL
LIN {X 0,Y 122.107,Z 1195.911,A -85,B 0,C 180,E1 31183.457,E2 31183.457} C_VEL
LIN {X 0,Y 102.427,Z 1187.807,A -85,B 0,C 180,E1 31208.439,E2 31208.439} C_VEL
LIN {X 0,Y 101.358,Z 1178.132,A -85,B 0,C 180,E1 31227.939,E2 31227.939} C_VEL
LIN {X 0,Y 101.121,Z 1165.977,A -85,B 0,C 180,E1 31241.957,E2 31241.957} C_VEL
LIN {X 0,Y 107.195,Z 1150.389,A -85,B 0,C 180,E1 31256.214,E2 31256.214} C_VEL
LIN {X 0,Y 117.808,Z 1157.076,A -85,B 0,C 180,E1 31273.608,E2 31273.608} C_VEL
LIN {X 0,Y 132.136,Z 1159.562,A -85,B 0,C 180,E1 31283.268,E2 31283.268} C_VEL
LIN {X 0,Y 139.149,Z 1159.683,A -85,B 0,C 180,E1 31287.121,E2 31287.121} C_VEL
LIN {X 0,Y 119.46,Z 1147.959,A -85,B 0,C 180,E1 31297.707,E2 31297.707} C_VEL
LIN {X 0,Y 106.368,Z 1129.834,A -85,B 0,C 180,E1 31311.842,E2 31311.842} C_VEL
LIN {X 0,Y 101.867,Z 1107.135,A -85,B 0,C 180,E1 31326.397,E2 31326.397} C_VEL
LIN {X 0,Y 102.138,Z 1080.924,A -85,B 0,C 180,E1 31338.333,E2 31338.333} C_VEL
LIN {X 0,Y 104.407,Z 1051.244,A -85,B 0,C 180,E1 31347.159,E2 31347.159} C_VEL
LIN {X 0,Y 106.882,Z 1018.47,A -85,B 0,C 180,E1 31352.843,E2 31352.843} C_VEL
LIN {X 0,Y 106.747,Z 999.913,A -85,B 0,C 180,E1 31355.081,E2 31355.081} C_VEL
LIN {X 0,Y 96.444,Z 948.084,A -85,B 0,C 180,E1 31362.105,E2 31362.105} C_VEL
LIN {X 0,Y 97.949,Z 941.904,A -85,B 0,C 180,E1 31365.872,E2 31365.872} C_VEL
LIN {X 0,Y 99.469,Z 936.308,A -85,B 0,C 180,E1 31367.516,E2 31367.516} C_VEL
LIN {X 0,Y 102.649,Z 938.989,A -85,B 0,C 180,E1 31383.209,E2 31383.209} C_VEL
LIN {X 0,Y 108.435,Z 946.42,A -85,B 0,C 180,E1 31395.233,E2 31395.233} C_VEL
LIN {X 0,Y 114.824,Z 955.178,A -85,B 0,C 180,E1 31404.033,E2 31404.033} C_VEL
LIN {X 0,Y 122.06,Z 976.962,A -85,B 0,C 180,E1 31414.595,E2 31414.595} C_VEL
LIN {X 0,Y 128.871,Z 1004.63,A -85,B 0,C 180,E1 31424.8,E2 31424.8} C_VEL
LIN {X 0,Y 134.609,Z 1037.014,A -85,B 0,C 180,E1 31435.351,E2 31435.351} C_VEL
LIN {X 0,Y 137.497,Z 1061.942,A -85,B 0,C 180,E1 31443.263,E2 31443.263} C_VEL
LIN {X 0,Y 120.753,Z 1098.496,A -85,B 0,C 180,E1 31453.503,E2 31453.503} C_VEL
LIN {X 0,Y 114.075,Z 1107.659,A -85,B 0,C 180,E1 31456.775,E2 31456.775} C_VEL
LIN {X 0,Y 102.883,Z 1120.216,A -85,B 0,C 180,E1 31462.38,E2 31462.38} C_VEL
LIN {X 0,Y 102.117,Z 1121.68,A -85,B 0,C 180,E1 31463.182,E2 31463.182} C_VEL
LIN {X 0,Y 93.337,Z 1145.727,A -85,B 0,C 180,E1 31479.867,E2 31479.867} C_VEL
LIN {X 0,Y 90.893,Z 1163.128,A -85,B 0,C 180,E1 31497.191,E2 31497.191} C_VEL
LIN {X 0,Y 92.673,Z 1175.719,A -85,B 0,C 180,E1 31514.147,E2 31514.147} C_VEL
LIN {X 0,Y 108.415,Z 1190.799,A -85,B 0,C 180,E1 31538.834,E2 31538.834} C_VEL
LIN {X 0,Y 112.596,Z 1192.789,A -85,B 0,C 180,E1 31542.135,E2 31542.135} C_VEL
LIN {X 0,Y 109.328,Z 1192.209,A -85,B 0,C 180,E1 31546.386,E2 31546.386} C_VEL
LIN {X 0,Y 94.255,Z 1183.477,A -85,B 0,C 180,E1 31571.385,E2 31571.385} C_VEL
LIN {X 0,Y 93.95,Z 1175.24,A -85,B 0,C 180,E1 31587.777,E2 31587.777} C_VEL
LIN {X 0,Y 93.669,Z 1162.454,A -85,B 0,C 180,E1 31603.017,E2 31603.017} C_VEL
LIN {X 0,Y 100.129,Z 1147.125,A -85,B 0,C 180,E1 31617.003,E2 31617.003} C_VEL
LIN {X 0,Y 117.859,Z 1155.503,A -85,B 0,C 180,E1 31640.383,E2 31640.383} C_VEL
LIN {X 0,Y 127.601,Z 1157.028,A -85,B 0,C 180,E1 31646.092,E2 31646.092} C_VEL
LIN {X 0,Y 125.974,Z 1155.667,A -85,B 0,C 180,E1 31648.016,E2 31648.016} C_VEL
LIN {X 0,Y 107.097,Z 1140.483,A -85,B 0,C 180,E1 31660.43,E2 31660.43} C_VEL
LIN {X 0,Y 96.8,Z 1120.279,A -85,B 0,C 180,E1 31675.533,E2 31675.533} C_VEL
LIN {X 0,Y 94.199,Z 1096.437,A -85,B 0,C 180,E1 31689.805,E2 31689.805} C_VEL
LIN {X 0,Y 95.136,Z 1069.74,A -85,B 0,C 180,E1 31700.95,E2 31700.95} C_VEL
LIN {X 0,Y 97.458,Z 1039.863,A -85,B 0,C 180,E1 31708.923,E2 31708.923} C_VEL
LIN {X 0,Y 99.366,Z 1003.074,A -85,B 0,C 180,E1 31714.496,E2 31714.496} C_VEL
LIN {X 0,Y 91.685,Z 965.514,A -85,B 0,C 180,E1 31719.596,E2 31719.596} C_VEL
LIN {X 0,Y 92.883,Z 960.286,A -85,B 0,C 180,E1 31723.559,E2 31723.559} C_VEL
LIN {X 0,Y 95.134,Z 952.223,A -85,B 0,C 180,E1 31726.745,E2 31726.745} C_VEL
LIN {X 0,Y 97.586,Z 944.361,A -85,B 0,C 180,E1 31730.751,E2 31730.751} C_VEL
LIN {X 0,Y 100.299,Z 946.542,A -85,B 0,C 180,E1 31742.619,E2 31742.619} C_VEL
LIN {X 0,Y 105.636,Z 953.898,A -85,B 0,C 180,E1 31754.65,E2 31754.65} C_VEL
LIN {X 0,Y 110.543,Z 960.878,A -85,B 0,C 180,E1 31762.074,E2 31762.074} C_VEL
LIN {X 0,Y 116.65,Z 980.779,A -85,B 0,C 180,E1 31772.435,E2 31772.435} C_VEL
LIN {X 0,Y 122.569,Z 1007.231,A -85,B 0,C 180,E1 31782.905,E2 31782.905} C_VEL
LIN {X 0,Y 127.584,Z 1038.833,A -85,B 0,C 180,E1 31793.869,E2 31793.869} C_VEL
LIN {X 0,Y 130.026,Z 1062.633,A -85,B 0,C 180,E1 31801.902,E2 31801.902} C_VEL
LIN {X 0,Y 112.787,Z 1098.956,A -85,B 0,C 180,E1 31812.614,E2 31812.614} C_VEL
LIN {X 0,Y 102.117,Z 1121.68,A -85,B 0,C 180,E1 31823.182,E2 31823.182} C_VEL
LIN {X 0,Y 93.668,Z 1132.235,A -85,B 0,C 180,E1 31829.734,E2 31829.734} C_VEL
LIN {X 0,Y 86.209,Z 1142.108,A -85,B 0,C 180,E1 31837.763,E2 31837.763} C_VEL
LIN {X 0,Y 83.284,Z 1160.508,A -85,B 0,C 180,E1 31856.934,E2 31856.934} C_VEL
LIN {X 0,Y 85.341,Z 1173.567,A -85,B 0,C 180,E1 31875.391,E2 31875.391} C_VEL
LIN {X 0,Y 101.252,Z 1188.491,A -85,B 0,C 180,E1 31900.469,E2 31900.469} C_VEL
LIN {X 0,Y 103.581,Z 1189.837,A -85,B 0,C 180,E1 31903.275,E2 31903.275} C_VEL
LIN {X 0,Y 87.238,Z 1180.747,A -85,B 0,C 180,E1 31929.826,E2 31929.826} C_VEL
LIN {X 0,Y 86.538,Z 1172.33,A -85,B 0,C 180,E1 31947.586,E2 31947.586} C_VEL
LIN {X 0,Y 86.457,Z 1157.783,A -85,B 0,C 180,E1 31965.391,E2 31965.391} C_VEL
LIN {X 0,Y 94.143,Z 1143.086,A -85,B 0,C 180,E1 31979.204,E2 31979.204} C_VEL
LIN {X 0,Y 113.244,Z 1152.506,A -85,B 0,C 180,E1 32003.295,E2 32003.295} C_VEL
LIN {X 0,Y 117.608,Z 1153.064,A -85,B 0,C 180,E1 32006.753,E2 32006.753} C_VEL
LIN {X 0,Y 98.867,Z 1136.375,A -85,B 0,C 180,E1 32019.896,E2 32019.896} C_VEL
LIN {X 0,Y 88.91,Z 1114.229,A -85,B 0,C 180,E1 32036.356,E2 32036.356} C_VEL
LIN {X 0,Y 86.802,Z 1090.134,A -85,B 0,C 180,E1 32050.649,E2 32050.649} C_VEL
LIN {X 0,Y 87.918,Z 1062.133,A -85,B 0,C 180,E1 32062.096,E2 32062.096} C_VEL
LIN {X 0,Y 90.218,Z 1031.528,A -85,B 0,C 180,E1 32069.83,E2 32069.83} C_VEL
LIN {X 0,Y 91.15,Z 1001.983,A -85,B 0,C 180,E1 32074.332,E2 32074.332} C_VEL
LIN {X 0,Y 86.874,Z 981.126,A -85,B 0,C 180,E1 32077.3,E2 32077.3} C_VEL
LIN {X 0,Y 87.765,Z 976.816,A -85,B 0,C 180,E1 32081.31,E2 32081.31} C_VEL
LIN {X 0,Y 89.629,Z 970.597,A -85,B 0,C 180,E1 32083.949,E2 32083.949} C_VEL
LIN {X 0,Y 92.849,Z 960.562,A -85,B 0,C 180,E1 32088.985,E2 32088.985} C_VEL
LIN {X 0,Y 95.783,Z 952.201,A -85,B 0,C 180,E1 32093.052,E2 32093.052} C_VEL
LIN {X 0,Y 97.877,Z 954.219,A -85,B 0,C 180,E1 32102.153,E2 32102.153} C_VEL
LIN {X 0,Y 102.82,Z 961.357,A -85,B 0,C 180,E1 32114.08,E2 32114.08} C_VEL
LIN {X 0,Y 107.325,Z 968.955,A -85,B 0,C 180,E1 32121.835,E2 32121.835} C_VEL
LIN {X 0,Y 112.546,Z 990.467,A -85,B 0,C 180,E1 32132.818,E2 32132.818} C_VEL
LIN {X 0,Y 117.154,Z 1015.397,A -85,B 0,C 180,E1 32142.977,E2 32142.977} C_VEL
LIN {X 0,Y 121.076,Z 1045.058,A -85,B 0,C 180,E1 32153.859,E2 32153.859} C_VEL
LIN {X 0,Y 122.64,Z 1063.218,A -85,B 0,C 180,E1 32160.387,E2 32160.387} C_VEL
LIN {X 0,Y 104.549,Z 1099.856,A -85,B 0,C 180,E1 32171.829,E2 32171.829} C_VEL
LIN {X 0,Y 90.463,Z 1130.005,A -85,B 0,C 180,E1 32188.246,E2 32188.246} C_VEL
LIN {X 0,Y 86.209,Z 1142.108,A -85,B 0,C 180,E1 32197.763,E2 32197.763} C_VEL
LIN {X 0,Y 81.911,Z 1149.076,A -85,B 0,C 180,E1 32204.776,E2 32204.776} C_VEL
LIN {X 0,Y 75.716,Z 1159.148,A -85,B 0,C 180,E1 32218.477,E2 32218.477} C_VEL
LIN {X 0,Y 78.915,Z 1172.823,A -85,B 0,C 180,E1 32239.566,E2 32239.566} C_VEL
LIN {X 0,Y 94.129,Z 1185.969,A -85,B 0,C 180,E1 32262.276,E2 32262.276} C_VEL
LIN {X 0,Y 92.911,Z 1185.82,A -85,B 0,C 180,E1 32265.453,E2 32265.453} C_VEL
LIN {X 0,Y 79.171,Z 1175.09,A -85,B 0,C 180,E1 32295.082,E2 32295.082} C_VEL
LIN {X 0,Y 79.17,Z 1169.127,A -85,B 0,C 180,E1 32307.362,E2 32307.362} C_VEL
LIN {X 0,Y 79.517,Z 1152.797,A -85,B 0,C 180,E1 32328.202,E2 32328.202} C_VEL
LIN {X 0,Y 88.527,Z 1139.012,A -85,B 0,C 180,E1 32341.974,E2 32341.974} C_VEL
LIN {X 0,Y 103.746,Z 1147.842,A -85,B 0,C 180,E1 32362.796,E2 32362.796} C_VEL
LIN {X 0,Y 108.059,Z 1149.001,A -85,B 0,C 180,E1 32365.999,E2 32365.999} C_VEL
LIN {X 0,Y 89.808,Z 1130.309,A -85,B 0,C 180,E1 32380.346,E2 32380.346} C_VEL
LIN {X 0,Y 81.107,Z 1107.439,A -85,B 0,C 180,E1 32397.342,E2 32397.342} C_VEL
LIN {X 0,Y 79.482,Z 1083.198,A -85,B 0,C 180,E1 32411.616,E2 32411.616} C_VEL
LIN {X 0,Y 80.863,Z 1053.42,A -85,B 0,C 180,E1 32423.409,E2 32423.409} C_VEL
LIN {X 0,Y 83.077,Z 1021.448,A -85,B 0,C 180,E1 32430.781,E2 32430.781} C_VEL
LIN {X 0,Y 83.121,Z 1001.895,A -85,B 0,C 180,E1 32433.891,E2 32433.891} C_VEL
LIN {X 0,Y 81.792,Z 995.75,A -85,B 0,C 180,E1 32435.153,E2 32435.153} C_VEL
LIN {X 0,Y 82.759,Z 991.15,A -85,B 0,C 180,E1 32439.526,E2 32439.526} C_VEL
LIN {X 0,Y 84.513,Z 985.655,A -85,B 0,C 180,E1 32442.407,E2 32442.407} C_VEL
LIN {X 0,Y 91.919,Z 965.21,A -85,B 0,C 180,E1 32453.023,E2 32453.023} C_VEL
LIN {X 0,Y 94.026,Z 959.972,A -85,B 0,C 180,E1 32455.468,E2 32455.468} C_VEL
LIN {X 0,Y 95.792,Z 963.044,A -85,B 0,C 180,E1 32463.531,E2 32463.531} C_VEL
LIN {X 0,Y 100.596,Z 969.879,A -85,B 0,C 180,E1 32475.026,E2 32475.026} C_VEL
LIN {X 0,Y 103.542,Z 976.319,A -85,B 0,C 180,E1 32480.96,E2 32480.96} C_VEL
LIN {X 0,Y 107.909,Z 998.304,A -85,B 0,C 180,E1 32492.437,E2 32492.437} C_VEL
LIN {X 0,Y 111.723,Z 1024.82,A -85,B 0,C 180,E1 32503.62,E2 32503.62} C_VEL
LIN {X 0,Y 114.858,Z 1055.609,A -85,B 0,C 180,E1 32515.591,E2 32515.591} C_VEL
LIN {X 0,Y 114.78,Z 1064.864,A -85,B 0,C 180,E1 32518.991,E2 32518.991} C_VEL
LIN {X 0,Y 96.311,Z 1100.699,A -85,B 0,C 180,E1 32530.954,E2 32530.954} C_VEL
LIN {X 0,Y 82.391,Z 1129.697,A -85,B 0,C 180,E1 32548.164,E2 32548.164} C_VEL
LIN {X 0,Y 76.109,Z 1152.439,A -85,B 0,C 180,E1 32570.029,E2 32570.029} C_VEL
LIN {X 0,Y 75.716,Z 1159.148,A -85,B 0,C 180,E1 32578.477,E2 32578.477} C_VEL
LIN {X 0,Y 73.873,Z 1164.534,A -85,B 0,C 180,E1 32587.533,E2 32587.533} C_VEL
LIN {X 0,Y 72.852,Z 1171.689,A -85,B 0,C 180,E1 32604.037,E2 32604.037} C_VEL
LIN {X 0,Y 85.477,Z 1182.182,A -85,B 0,C 180,E1 32622.751,E2 32622.751} C_VEL
LIN {X 0,Y 83.601,Z 1181.649,A -85,B 0,C 180,E1 32626.287,E2 32626.287} C_VEL
LIN {X 0,Y 71.89,Z 1170.328,A -85,B 0,C 180,E1 32657.976,E2 32657.976} C_VEL
LIN {X 0,Y 71.786,Z 1165.871,A -85,B 0,C 180,E1 32667.09,E2 32667.09} C_VEL
LIN {X 0,Y 75.646,Z 1142.774,A -85,B 0,C 180,E1 32696.819,E2 32696.819} C_VEL
LIN {X 0,Y 82.94,Z 1135.017,A -85,B 0,C 180,E1 32704.813,E2 32704.813} C_VEL
LIN {X 0,Y 95.212,Z 1142.811,A -85,B 0,C 180,E1 32722.642,E2 32722.642} C_VEL
LIN {X 0,Y 97.543,Z 1143.14,A -85,B 0,C 180,E1 32725.919,E2 32725.919} C_VEL
LIN {X 0,Y 80.529,Z 1122.565,A -85,B 0,C 180,E1 32741.595,E2 32741.595} C_VEL
